// TwinCAT 3 PLC project LeakTesters
// ProgramVersion: 3.1.4024.0
// libraries:
//   Tc2_Standard, * (Beckhoff Automation GmbH)
//   Tc2_System, * (Beckhoff Automation GmbH)
//   Tc2_Utilities, * (Beckhoff Automation GmbH)
//   Tc3_EventLogger, * (Beckhoff Automation GmbH)
//   Tc3_Module, * (Beckhoff Automation GmbH)
//   VisuUserMgmt, * (System)
// project tree:
//   DUTs/ E_MachineState.TcDUT (not stored), E_StationState.TcDUT (not stored), ST_ActiveEventsHMI.TcDUT (not stored), ST_AlarmHistory.TcDUT (not stored), ST_Events.TcDUT (not stored), ST_HeightLimits.TcDUT (not stored), ST_HeightMeasurement2.TcDUT (not stored), ST_MachineStatusStruct.TcDUT (not stored), ST_MasterControlStruct.TcDUT (not stored), ST_MeasureStatistics.TcDUT (not stored), ST_Nest.TcDUT, ST_PartsInspection.TcDUT, ST_StandardStationStruct.TcDUT (not stored), ST_UserLogHMI.TcDUT (not stored)
//   DUTs/HeightMeasureFunction/ E_HeighttMeasureProcess.TcDUT (not stored)
//   DUTs/IO/ E_BoxDiag.TcDUT (not stored), E_BoxState.TcDUT (not stored), E_TerminalState.TcDUT (not stored), st_Box_Info.TcDUT (not stored), st_EL1809.TcDUT (not stored), st_EL2809.TcDUT (not stored), ST_DL_PN1.TcDUT (not stored), st_KeyenceCamera.TcDUT, st_Terminal_Info.TcDUT (not stored)
//   GVLs/ GVL_Constants.TcGVL (not stored), GVL_HMI_GLOBAL.TcGVL, GVL_IO.TcGVL, GVL_MASTER.TcGVL (not stored), GVL_PERSIST.TcGVL
//   / PlcTask.TcTTO (not stored)
//   POUs/A_Master/ Main_Master.TcPOU, PRG_FaultHandling.TcPOU, PRG_MachineStatus.TcPOU (not stored), PRG_MasterCycle.TcPOU, PRG_MasterSystemTime.TcPOU (not stored), PRG_TerminBoxInfo.TcPOU (not stored)
//   POUs/B_HightTest/ PRG_Fault_HeightTest.TcPOU (not stored), PRG_HeightTest.TcPOU
//   POUs/D_VisionTest/ PRG_Fault_VisionTest.TcPOU, PRG_VisionTest.TcPOU
//   POUs/E_HMI/ PRG_HMI.TcPOU
//   POUs/G_Utility/ FB_Alarms.TcPOU (not stored), FB_BoxInfo.TcPOU (not stored), FB_DayOfYear.TcPOU (not stored), FB_EventLog.TcPOU (not stored), FB_HeightMeasurement2.TcPOU (not stored), FB_Pulse.TcPOU (not stored), FB_TerminalInfo.TcPOU (not stored), FB_TimeControl.TcPOU (not stored), PRG_Puls.TcPOU (not stored)
//   POUs/ MAIN.TcPOU (not stored)
// real-time tasks:
//   TASK PlcTask: cycle T#10ms, priority 20, ADS port 350
// I/O:
//   DEVICE Device 1 (EtherCAT), AmsNetId 172.18.239.139.2.1
//     Term 9 (EK1100) [EK1100 EtherCAT Coupler (2A E-Bus)]
//       Term 10 (EL6070-0033) [EL6070-0033 1Ch. Licence key terminal, individual licences]
//       Term 11 (EL1809) [EL1809 16Ch. Dig. Input 24V, 3ms]
//       Term 12 (EL2809-0015) [EL2809-0015 16Ch. Dig. Output 24V DC, 0.35A, not short-circuit proof]
//       Term 13 (EL6631) [EL6631 PROFINET IO Controller]
//       Term 14 (EL9011) [EL9011 End Terminal]
//   DEVICE Device 2 (EL6631), AmsNetId 172.18.239.139.3.1
//     dl-pn1 [Keyence DL-PN1 PROFINET IO Device DL-PN1]
//       modules: Term 13 (DAP Module), Term 14 (DL-PN1), Term 15 (GT2-1.1), Term 16 (GT2-1.2), Term 17 (GT2-1.3), Term 18 (GT2-2)
//     camera-1 [KEYENCE CORPORATION. IV4-XXXX IV4-XXXX]
//       modules: Term 1 (DAP Module), Term 2 (Command Control), Term 3 (Additional Setting Value), Term 4 (Command Status Bits), Term 5 (Device Result Bits), Term 6 (Device Status Words), Term 7 (Device Statistics), Term 8 (Position Adjust Result), Term 9 (Tool Result), Term 10 (Tool Result), Term 11 (Tool Result), Term 79 (Device Result Bits)
// variable links:
//   LeakTesters/LeakTesters Instance <-> Device 1 (EtherCAT)/Term 9 (EK1100)/Term 10 (EL6070-0033)
//     PlcTask Inputs/GVL_IO.dwTerminalInfo[2].nTerminal_State <-> InfoData/State
//   LeakTesters/LeakTesters Instance <-> Device 1 (EtherCAT)/Term 9 (EK1100)/Term 11 (EL1809)
//     PlcTask Inputs/GVL_IO.dwTerminalInfo[3].nTerminal_State <-> InfoData/State
//     PlcTask Inputs/GVL_IO.dw_T02_EL1809.iCalmpClosed <-> Channel 1/Input
//     PlcTask Inputs/GVL_IO.dw_T02_EL1809.iPartPresent <-> Channel 2/Input
//   LeakTesters/LeakTesters Instance <-> Device 1 (EtherCAT)/Term 9 (EK1100)/Term 12 (EL2809-0015)
//     PlcTask Inputs/GVL_IO.dwTerminalInfo[4].nTerminal_State <-> InfoData/State
//     PlcTask Outputs/GVL_IO.dw_T03_EL2809.qEL2809_Ch3 <-> Channel 3/Output
//     PlcTask Outputs/GVL_IO.dw_T03_EL2809.qPassIndicatorGreen <-> Channel 1/Output
//     PlcTask Outputs/GVL_IO.dw_T03_EL2809.qRejectIndicatorRed <-> Channel 2/Output
//   LeakTesters/LeakTesters Instance <-> Device 1 (EtherCAT)/Term 9 (EK1100)/Term 13 (EL6631)
//     PlcTask Inputs/GVL_IO.dwTerminalInfo[5].nTerminal_State <-> InfoData/State
//   LeakTesters/LeakTesters Instance <-> Device 2 (EL6631)/camera-1
//     PlcTask Inputs/GVL_IO.dw_B06_KeyenceCamera.bBusy <-> API/Term 4 (Command Status Bits)/Subterm 6 (Command Status Bits)/Inputs/Command Status Bits Register2/Busy
//     PlcTask Inputs/GVL_IO.dw_B06_KeyenceCamera.bError <-> API/Term 4 (Command Status Bits)/Subterm 6 (Command Status Bits)/Inputs/Command Status Bits Register3/Error
//     PlcTask Inputs/GVL_IO.dw_B06_KeyenceCamera.bReady <-> API/Term 4 (Command Status Bits)/Subterm 6 (Command Status Bits)/Inputs/Command Status Bits Register2/Ready
//     PlcTask Inputs/GVL_IO.dw_B06_KeyenceCamera.bResultReady <-> API/Term 4 (Command Status Bits)/Subterm 6 (Command Status Bits)/Inputs/Command Status Bits Register2/Result_Ready
//     PlcTask Inputs/GVL_IO.dw_B06_KeyenceCamera.bRun <-> API/Term 4 (Command Status Bits)/Subterm 6 (Command Status Bits)/Inputs/Command Status Bits Register2/Run
//     PlcTask Inputs/GVL_IO.dw_B06_KeyenceCamera.bTotalResult <-> API/Term 5 (Device Result Bits)/Subterm 7 (Device Result Bits)/Inputs/Device Result Bits Register0/Total_Status
//     PlcTask Inputs/GVL_IO.dw_B06_KeyenceCamera.bTriggerFail <-> API/Term 4 (Command Status Bits)/Subterm 6 (Command Status Bits)/Inputs/Command Status Bits Register1/Trigger_Fail
//     PlcTask Outputs/GVL_IO.dw_B06_KeyenceCamera.bClearBuffer <-> API/Term 2 (Command Control)/Subterm 4 (Command Control)/Outputs/Command Control Register0/Clear_Buffer
//     PlcTask Outputs/GVL_IO.dw_B06_KeyenceCamera.bReset <-> API/Term 2 (Command Control)/Subterm 4 (Command Control)/Outputs/Command Control Register0/Clear_Warning
//     PlcTask Outputs/GVL_IO.dw_B06_KeyenceCamera.bResultReadyAck <-> API/Term 2 (Command Control)/Subterm 4 (Command Control)/Outputs/Command Control Register1/Result_Ready_Ack
//     PlcTask Outputs/GVL_IO.dw_B06_KeyenceCamera.bTrigger <-> API/Term 2 (Command Control)/Subterm 4 (Command Control)/Outputs/Command Control Register0/Trigger
//   LeakTesters/LeakTesters Instance <-> Device 2 (EL6631)/dl-pn1
//     PlcTask Inputs/GVL_IO.dwBoxInfo[17].nPnIoBoxDiag <-> Inputs/PnIoBoxDiag
//     PlcTask Inputs/GVL_IO.dwBoxInfo[17].nPnIoBoxState <-> Inputs/PnIoBoxState
//     PlcTask Inputs/GVL_IO.dw_B08_DL_PN1.dldCurrValProp <-> API/Term 14 (DL-PN1)/Subterm 23 (DL-PN1 Device)/Inputs/Sensors Status/Current_Value_Property
//     PlcTask Inputs/GVL_IO.dw_B08_DL_PN1.dldErrorStt <-> API/Term 14 (DL-PN1)/Subterm 23 (DL-PN1 Device)/Inputs/Sensors Status/Error_Status
//     PlcTask Inputs/GVL_IO.dw_B08_DL_PN1.dldExtInpResp[1] <-> API/Term 14 (DL-PN1)/Subterm 23 (DL-PN1 Device)/Inputs/External Input Response/External_Input_Response_1
//     PlcTask Inputs/GVL_IO.dw_B08_DL_PN1.dldExtInpResp[2] <-> API/Term 14 (DL-PN1)/Subterm 23 (DL-PN1 Device)/Inputs/External Input Response/External_Input_Response_2
//     PlcTask Inputs/GVL_IO.dw_B08_DL_PN1.dldExtInpResp[3] <-> API/Term 14 (DL-PN1)/Subterm 23 (DL-PN1 Device)/Inputs/External Input Response/External_Input_Response_3
//     PlcTask Inputs/GVL_IO.dw_B08_DL_PN1.dldExtInpResp[4] <-> API/Term 14 (DL-PN1)/Subterm 23 (DL-PN1 Device)/Inputs/External Input Response/External_Input_Response_4
//     PlcTask Inputs/GVL_IO.dw_B08_DL_PN1.dldExtInpResp[5] <-> API/Term 14 (DL-PN1)/Subterm 23 (DL-PN1 Device)/Inputs/External Input Response/External_Input_Response_5
//     PlcTask Inputs/GVL_IO.dw_B08_DL_PN1.dldWarningStat <-> API/Term 14 (DL-PN1)/Subterm 23 (DL-PN1 Device)/Inputs/Sensors Status/Warning_Status
//     PlcTask Inputs/GVL_IO.dw_B08_DL_PN1.gt2_1_1CurrValInv <-> API/Term 15 (GT2-1.1)/Subterm 24 (GT2-***)/Inputs/Sensor Status/Current_Value_Invalid
//     PlcTask Inputs/GVL_IO.dw_B08_DL_PN1.gt2_1_2CurrValInv <-> API/Term 16 (GT2-1.2)/Subterm 25 (GT2-***)/Inputs/Sensor Status/Current_Value_Invalid
//     PlcTask Inputs/GVL_IO.dw_B08_DL_PN1.gt2_1_3CurrValInv <-> API/Term 17 (GT2-1.3)/Subterm 26 (GT2-***)/Inputs/Sensor Status/Current_Value_Invalid
//     PlcTask Inputs/GVL_IO.dw_B08_DL_PN1.gt2_1_1CurrValOvrR <-> API/Term 15 (GT2-1.1)/Subterm 24 (GT2-***)/Inputs/Sensor Status/Current_Value_Over_Range
//     PlcTask Inputs/GVL_IO.dw_B08_DL_PN1.gt2_1_2CurrValOvrR <-> API/Term 16 (GT2-1.2)/Subterm 25 (GT2-***)/Inputs/Sensor Status/Current_Value_Over_Range
//     PlcTask Inputs/GVL_IO.dw_B08_DL_PN1.gt2_1_3CurrValOvrR <-> API/Term 17 (GT2-1.3)/Subterm 26 (GT2-***)/Inputs/Sensor Status/Current_Value_Over_Range
//     PlcTask Inputs/GVL_IO.dw_B08_DL_PN1.gt2_1_1CurrValUndR <-> API/Term 15 (GT2-1.1)/Subterm 24 (GT2-***)/Inputs/Sensor Status/Current_Value_Under_Range
//     PlcTask Inputs/GVL_IO.dw_B08_DL_PN1.gt2_1_2CurrValUndR <-> API/Term 16 (GT2-1.2)/Subterm 25 (GT2-***)/Inputs/Sensor Status/Current_Value_Under_Range
//     PlcTask Inputs/GVL_IO.dw_B08_DL_PN1.gt2_1_3CurrValUndR <-> API/Term 17 (GT2-1.3)/Subterm 26 (GT2-***)/Inputs/Sensor Status/Current_Value_Under_Range
//     PlcTask Inputs/GVL_IO.dw_B08_DL_PN1.gt2_1_1CurrentValue <-> API/Term 15 (GT2-1.1)/Subterm 24 (GT2-***)/Inputs/Current Value
//     PlcTask Inputs/GVL_IO.dw_B08_DL_PN1.gt2_1_2CurrentValue <-> API/Term 16 (GT2-1.2)/Subterm 25 (GT2-***)/Inputs/Current Value
//     PlcTask Inputs/GVL_IO.dw_B08_DL_PN1.gt2_1_3CurrentValue <-> API/Term 17 (GT2-1.3)/Subterm 26 (GT2-***)/Inputs/Current Value
//     PlcTask Inputs/GVL_IO.dw_B08_DL_PN1.gt2_1_1ErrorStat <-> API/Term 15 (GT2-1.1)/Subterm 24 (GT2-***)/Inputs/Sensor Status/Error_Status
//     PlcTask Inputs/GVL_IO.dw_B08_DL_PN1.gt2_1_2ErrorStat <-> API/Term 16 (GT2-1.2)/Subterm 25 (GT2-***)/Inputs/Sensor Status/Error_Status
//     PlcTask Inputs/GVL_IO.dw_B08_DL_PN1.gt2_1_3ErrorStat <-> API/Term 17 (GT2-1.3)/Subterm 26 (GT2-***)/Inputs/Sensor Status/Error_Status
//     PlcTask Inputs/GVL_IO.dw_B08_DL_PN1.gt2_1_1ExtInpRes[1] <-> API/Term 15 (GT2-1.1)/Subterm 24 (GT2-***)/Inputs/External Input Response/External_Input_Response_1
//     PlcTask Inputs/GVL_IO.dw_B08_DL_PN1.gt2_1_1ExtInpRes[2] <-> API/Term 15 (GT2-1.1)/Subterm 24 (GT2-***)/Inputs/External Input Response/External_Input_Response_2
//     PlcTask Inputs/GVL_IO.dw_B08_DL_PN1.gt2_1_1ExtInpRes[3] <-> API/Term 15 (GT2-1.1)/Subterm 24 (GT2-***)/Inputs/External Input Response/External_Input_Response_3
//     PlcTask Inputs/GVL_IO.dw_B08_DL_PN1.gt2_1_1ExtInpRes[4] <-> API/Term 15 (GT2-1.1)/Subterm 24 (GT2-***)/Inputs/External Input Response/External_Input_Response_4
//     PlcTask Inputs/GVL_IO.dw_B08_DL_PN1.gt2_1_1ExtInpRes[5] <-> API/Term 15 (GT2-1.1)/Subterm 24 (GT2-***)/Inputs/External Input Response/External_Input_Response_5
//     PlcTask Inputs/GVL_IO.dw_B08_DL_PN1.gt2_1_2ExtInpRes[1] <-> API/Term 16 (GT2-1.2)/Subterm 25 (GT2-***)/Inputs/External Input Response/External_Input_Response_1
//     PlcTask Inputs/GVL_IO.dw_B08_DL_PN1.gt2_1_2ExtInpRes[2] <-> API/Term 16 (GT2-1.2)/Subterm 25 (GT2-***)/Inputs/External Input Response/External_Input_Response_2
//     PlcTask Inputs/GVL_IO.dw_B08_DL_PN1.gt2_1_2ExtInpRes[3] <-> API/Term 16 (GT2-1.2)/Subterm 25 (GT2-***)/Inputs/External Input Response/External_Input_Response_3
//     PlcTask Inputs/GVL_IO.dw_B08_DL_PN1.gt2_1_2ExtInpRes[4] <-> API/Term 16 (GT2-1.2)/Subterm 25 (GT2-***)/Inputs/External Input Response/External_Input_Response_4
//     PlcTask Inputs/GVL_IO.dw_B08_DL_PN1.gt2_1_2ExtInpRes[5] <-> API/Term 16 (GT2-1.2)/Subterm 25 (GT2-***)/Inputs/External Input Response/External_Input_Response_5
//     PlcTask Inputs/GVL_IO.dw_B08_DL_PN1.gt2_1_3ExtInpRes[1] <-> API/Term 17 (GT2-1.3)/Subterm 26 (GT2-***)/Inputs/External Input Response/External_Input_Response_1
//     PlcTask Inputs/GVL_IO.dw_B08_DL_PN1.gt2_1_3ExtInpRes[2] <-> API/Term 17 (GT2-1.3)/Subterm 26 (GT2-***)/Inputs/External Input Response/External_Input_Response_2
//     PlcTask Inputs/GVL_IO.dw_B08_DL_PN1.gt2_1_3ExtInpRes[3] <-> API/Term 17 (GT2-1.3)/Subterm 26 (GT2-***)/Inputs/External Input Response/External_Input_Response_3
//     PlcTask Inputs/GVL_IO.dw_B08_DL_PN1.gt2_1_3ExtInpRes[4] <-> API/Term 17 (GT2-1.3)/Subterm 26 (GT2-***)/Inputs/External Input Response/External_Input_Response_4
//     PlcTask Inputs/GVL_IO.dw_B08_DL_PN1.gt2_1_3ExtInpRes[5] <-> API/Term 17 (GT2-1.3)/Subterm 26 (GT2-***)/Inputs/External Input Response/External_Input_Response_5
//     PlcTask Inputs/GVL_IO.dw_B08_DL_PN1.gt2_1_1Output[1] <-> API/Term 15 (GT2-1.1)/Subterm 24 (GT2-***)/Inputs/Sensor Outputs/Output_1
//     PlcTask Inputs/GVL_IO.dw_B08_DL_PN1.gt2_1_1Output[2] <-> API/Term 15 (GT2-1.1)/Subterm 24 (GT2-***)/Inputs/Sensor Outputs/Output_2
//     PlcTask Inputs/GVL_IO.dw_B08_DL_PN1.gt2_1_1Output[3] <-> API/Term 15 (GT2-1.1)/Subterm 24 (GT2-***)/Inputs/Sensor Outputs/Output_3
//     PlcTask Inputs/GVL_IO.dw_B08_DL_PN1.gt2_1_1Output[4] <-> API/Term 15 (GT2-1.1)/Subterm 24 (GT2-***)/Inputs/Sensor Outputs/Output_4
//     PlcTask Inputs/GVL_IO.dw_B08_DL_PN1.gt2_1_1Output[5] <-> API/Term 15 (GT2-1.1)/Subterm 24 (GT2-***)/Inputs/Sensor Outputs/Output_5
//     PlcTask Inputs/GVL_IO.dw_B08_DL_PN1.gt2_1_2Output[1] <-> API/Term 16 (GT2-1.2)/Subterm 25 (GT2-***)/Inputs/Sensor Outputs/Output_1
//     PlcTask Inputs/GVL_IO.dw_B08_DL_PN1.gt2_1_2Output[2] <-> API/Term 16 (GT2-1.2)/Subterm 25 (GT2-***)/Inputs/Sensor Outputs/Output_2
//     PlcTask Inputs/GVL_IO.dw_B08_DL_PN1.gt2_1_2Output[3] <-> API/Term 16 (GT2-1.2)/Subterm 25 (GT2-***)/Inputs/Sensor Outputs/Output_3
//     PlcTask Inputs/GVL_IO.dw_B08_DL_PN1.gt2_1_2Output[4] <-> API/Term 16 (GT2-1.2)/Subterm 25 (GT2-***)/Inputs/Sensor Outputs/Output_4
//     PlcTask Inputs/GVL_IO.dw_B08_DL_PN1.gt2_1_2Output[5] <-> API/Term 16 (GT2-1.2)/Subterm 25 (GT2-***)/Inputs/Sensor Outputs/Output_5
//     PlcTask Inputs/GVL_IO.dw_B08_DL_PN1.gt2_1_3Output[1] <-> API/Term 17 (GT2-1.3)/Subterm 26 (GT2-***)/Inputs/Sensor Outputs/Output_1
//     PlcTask Inputs/GVL_IO.dw_B08_DL_PN1.gt2_1_3Output[2] <-> API/Term 17 (GT2-1.3)/Subterm 26 (GT2-***)/Inputs/Sensor Outputs/Output_2
//     PlcTask Inputs/GVL_IO.dw_B08_DL_PN1.gt2_1_3Output[3] <-> API/Term 17 (GT2-1.3)/Subterm 26 (GT2-***)/Inputs/Sensor Outputs/Output_3
//     PlcTask Inputs/GVL_IO.dw_B08_DL_PN1.gt2_1_3Output[4] <-> API/Term 17 (GT2-1.3)/Subterm 26 (GT2-***)/Inputs/Sensor Outputs/Output_4
//     PlcTask Inputs/GVL_IO.dw_B08_DL_PN1.gt2_1_3Output[5] <-> API/Term 17 (GT2-1.3)/Subterm 26 (GT2-***)/Inputs/Sensor Outputs/Output_5
//     PlcTask Inputs/GVL_IO.dw_B08_DL_PN1.gt2_1_1WarningStat <-> API/Term 15 (GT2-1.1)/Subterm 24 (GT2-***)/Inputs/Sensor Status/Warning_Status
//     PlcTask Inputs/GVL_IO.dw_B08_DL_PN1.gt2_1_2WarningStat <-> API/Term 16 (GT2-1.2)/Subterm 25 (GT2-***)/Inputs/Sensor Status/Warning_Status
//     PlcTask Inputs/GVL_IO.dw_B08_DL_PN1.gt2_1_3WarningStat <-> API/Term 17 (GT2-1.3)/Subterm 26 (GT2-***)/Inputs/Sensor Status/Warning_Status
//     PlcTask Inputs/GVL_IO.dw_B08_DL_PN1.gt2_2CurrValInv <-> API/Term 18 (GT2-2)/Subterm 27 (GT2-***)/Inputs/Sensor Status/Current_Value_Invalid
//     PlcTask Inputs/GVL_IO.dw_B08_DL_PN1.gt2_2CurrValOvrR <-> API/Term 18 (GT2-2)/Subterm 27 (GT2-***)/Inputs/Sensor Status/Current_Value_Over_Range
//     PlcTask Inputs/GVL_IO.dw_B08_DL_PN1.gt2_2CurrValUndR <-> API/Term 18 (GT2-2)/Subterm 27 (GT2-***)/Inputs/Sensor Status/Current_Value_Under_Range
//     PlcTask Inputs/GVL_IO.dw_B08_DL_PN1.gt2_2CurrentValue <-> API/Term 18 (GT2-2)/Subterm 27 (GT2-***)/Inputs/Current Value
//     PlcTask Inputs/GVL_IO.dw_B08_DL_PN1.gt2_2ErrorStat <-> API/Term 18 (GT2-2)/Subterm 27 (GT2-***)/Inputs/Sensor Status/Error_Status
//     PlcTask Inputs/GVL_IO.dw_B08_DL_PN1.gt2_2ExtInpRes[1] <-> API/Term 18 (GT2-2)/Subterm 27 (GT2-***)/Inputs/External Input Response/External_Input_Response_1
//     PlcTask Inputs/GVL_IO.dw_B08_DL_PN1.gt2_2ExtInpRes[2] <-> API/Term 18 (GT2-2)/Subterm 27 (GT2-***)/Inputs/External Input Response/External_Input_Response_2
//     PlcTask Inputs/GVL_IO.dw_B08_DL_PN1.gt2_2ExtInpRes[3] <-> API/Term 18 (GT2-2)/Subterm 27 (GT2-***)/Inputs/External Input Response/External_Input_Response_3
//     PlcTask Inputs/GVL_IO.dw_B08_DL_PN1.gt2_2ExtInpRes[4] <-> API/Term 18 (GT2-2)/Subterm 27 (GT2-***)/Inputs/External Input Response/External_Input_Response_4
//     PlcTask Inputs/GVL_IO.dw_B08_DL_PN1.gt2_2ExtInpRes[5] <-> API/Term 18 (GT2-2)/Subterm 27 (GT2-***)/Inputs/External Input Response/External_Input_Response_5
//     PlcTask Inputs/GVL_IO.dw_B08_DL_PN1.gt2_2Output[1] <-> API/Term 18 (GT2-2)/Subterm 27 (GT2-***)/Inputs/Sensor Outputs/Output_1
//     PlcTask Inputs/GVL_IO.dw_B08_DL_PN1.gt2_2Output[2] <-> API/Term 18 (GT2-2)/Subterm 27 (GT2-***)/Inputs/Sensor Outputs/Output_2
//     PlcTask Inputs/GVL_IO.dw_B08_DL_PN1.gt2_2Output[3] <-> API/Term 18 (GT2-2)/Subterm 27 (GT2-***)/Inputs/Sensor Outputs/Output_3
//     PlcTask Inputs/GVL_IO.dw_B08_DL_PN1.gt2_2Output[4] <-> API/Term 18 (GT2-2)/Subterm 27 (GT2-***)/Inputs/Sensor Outputs/Output_4
//     PlcTask Inputs/GVL_IO.dw_B08_DL_PN1.gt2_2Output[5] <-> API/Term 18 (GT2-2)/Subterm 27 (GT2-***)/Inputs/Sensor Outputs/Output_5
//     PlcTask Inputs/GVL_IO.dw_B08_DL_PN1.gt2_2WarningStat <-> API/Term 18 (GT2-2)/Subterm 27 (GT2-***)/Inputs/Sensor Status/Warning_Status
//     PlcTask Outputs/GVL_IO.dw_B08_DL_PN1.dldExtInpRespOut[1] <-> API/Term 14 (DL-PN1)/Subterm 23 (DL-PN1 Device)/Outputs/External Input Requests/External_Input_Request_1
//     PlcTask Outputs/GVL_IO.dw_B08_DL_PN1.dldExtInpRespOut[2] <-> API/Term 14 (DL-PN1)/Subterm 23 (DL-PN1 Device)/Outputs/External Input Requests/External_Input_Request_2
//     PlcTask Outputs/GVL_IO.dw_B08_DL_PN1.dldExtInpRespOut[3] <-> API/Term 14 (DL-PN1)/Subterm 23 (DL-PN1 Device)/Outputs/External Input Requests/External_Input_Request_3
//     PlcTask Outputs/GVL_IO.dw_B08_DL_PN1.dldExtInpRespOut[4] <-> API/Term 14 (DL-PN1)/Subterm 23 (DL-PN1 Device)/Outputs/External Input Requests/External_Input_Request_4
//     PlcTask Outputs/GVL_IO.dw_B08_DL_PN1.dldExtInpRespOut[5] <-> API/Term 14 (DL-PN1)/Subterm 23 (DL-PN1 Device)/Outputs/External Input Requests/External_Input_Request_5
//     PlcTask Outputs/GVL_IO.dw_B08_DL_PN1.gt2_1_1ExtInpResOut[1] <-> API/Term 15 (GT2-1.1)/Subterm 24 (GT2-***)/Outputs/External Input Requests/External_Input_Request_1
//     PlcTask Outputs/GVL_IO.dw_B08_DL_PN1.gt2_1_1ExtInpResOut[2] <-> API/Term 15 (GT2-1.1)/Subterm 24 (GT2-***)/Outputs/External Input Requests/External_Input_Request_2
//     PlcTask Outputs/GVL_IO.dw_B08_DL_PN1.gt2_1_1ExtInpResOut[3] <-> API/Term 15 (GT2-1.1)/Subterm 24 (GT2-***)/Outputs/External Input Requests/External_Input_Request_3
//     PlcTask Outputs/GVL_IO.dw_B08_DL_PN1.gt2_1_1ExtInpResOut[4] <-> API/Term 15 (GT2-1.1)/Subterm 24 (GT2-***)/Outputs/External Input Requests/External_Input_Request_4
//     PlcTask Outputs/GVL_IO.dw_B08_DL_PN1.gt2_1_1ExtInpResOut[5] <-> API/Term 15 (GT2-1.1)/Subterm 24 (GT2-***)/Outputs/External Input Requests/External_Input_Request_5
//     PlcTask Outputs/GVL_IO.dw_B08_DL_PN1.gt2_1_2ExtInpResOut[1] <-> API/Term 16 (GT2-1.2)/Subterm 25 (GT2-***)/Outputs/External Input Requests/External_Input_Request_1
//     PlcTask Outputs/GVL_IO.dw_B08_DL_PN1.gt2_1_2ExtInpResOut[2] <-> API/Term 16 (GT2-1.2)/Subterm 25 (GT2-***)/Outputs/External Input Requests/External_Input_Request_2
//     PlcTask Outputs/GVL_IO.dw_B08_DL_PN1.gt2_1_2ExtInpResOut[3] <-> API/Term 16 (GT2-1.2)/Subterm 25 (GT2-***)/Outputs/External Input Requests/External_Input_Request_3
//     PlcTask Outputs/GVL_IO.dw_B08_DL_PN1.gt2_1_2ExtInpResOut[4] <-> API/Term 16 (GT2-1.2)/Subterm 25 (GT2-***)/Outputs/External Input Requests/External_Input_Request_4
//     PlcTask Outputs/GVL_IO.dw_B08_DL_PN1.gt2_1_2ExtInpResOut[5] <-> API/Term 16 (GT2-1.2)/Subterm 25 (GT2-***)/Outputs/External Input Requests/External_Input_Request_5
//     PlcTask Outputs/GVL_IO.dw_B08_DL_PN1.gt2_1_3ExtInpResOut[1] <-> API/Term 17 (GT2-1.3)/Subterm 26 (GT2-***)/Outputs/External Input Requests/External_Input_Request_1
//     PlcTask Outputs/GVL_IO.dw_B08_DL_PN1.gt2_1_3ExtInpResOut[2] <-> API/Term 17 (GT2-1.3)/Subterm 26 (GT2-***)/Outputs/External Input Requests/External_Input_Request_2
//     PlcTask Outputs/GVL_IO.dw_B08_DL_PN1.gt2_1_3ExtInpResOut[3] <-> API/Term 17 (GT2-1.3)/Subterm 26 (GT2-***)/Outputs/External Input Requests/External_Input_Request_3
//     PlcTask Outputs/GVL_IO.dw_B08_DL_PN1.gt2_1_3ExtInpResOut[4] <-> API/Term 17 (GT2-1.3)/Subterm 26 (GT2-***)/Outputs/External Input Requests/External_Input_Request_4
//     PlcTask Outputs/GVL_IO.dw_B08_DL_PN1.gt2_1_3ExtInpResOut[5] <-> API/Term 17 (GT2-1.3)/Subterm 26 (GT2-***)/Outputs/External Input Requests/External_Input_Request_5
//     PlcTask Outputs/GVL_IO.dw_B08_DL_PN1.gt2_2ExtInpResOut[1] <-> API/Term 18 (GT2-2)/Subterm 27 (GT2-***)/Outputs/External Input Requests/External_Input_Request_1
//     PlcTask Outputs/GVL_IO.dw_B08_DL_PN1.gt2_2ExtInpResOut[2] <-> API/Term 18 (GT2-2)/Subterm 27 (GT2-***)/Outputs/External Input Requests/External_Input_Request_2
//     PlcTask Outputs/GVL_IO.dw_B08_DL_PN1.gt2_2ExtInpResOut[3] <-> API/Term 18 (GT2-2)/Subterm 27 (GT2-***)/Outputs/External Input Requests/External_Input_Request_3
//     PlcTask Outputs/GVL_IO.dw_B08_DL_PN1.gt2_2ExtInpResOut[4] <-> API/Term 18 (GT2-2)/Subterm 27 (GT2-***)/Outputs/External Input Requests/External_Input_Request_4
//     PlcTask Outputs/GVL_IO.dw_B08_DL_PN1.gt2_2ExtInpResOut[5] <-> API/Term 18 (GT2-2)/Subterm 27 (GT2-***)/Outputs/External Input Requests/External_Input_Request_5

// ---- DUTs/IO/st_KeyenceCamera.TcDUT
TYPE st_KeyenceCamera :
STRUCT
	
	////////////////////////////////////////////////////INPUTS//////////////////////////////////////////////////

	bResultReady							AT%I*					: BOOL;
	bError									AT%I*					: BOOL;
	bBusy									AT%I*					: BOOL;
	bRun									AT%I*					: BOOL;
	bReady									AT%I*					: BOOL;
	bTotalResult							AT%I*					: BOOL;
	bTriggerFail							AT%I*					: BOOL;
	
	////////////////////////////////////////////////////OUTPUTS//////////////////////////////////////////////////
	
	bTrigger								AT%Q*					: BOOL;//
	bReset									AT%Q*					: BOOL;//
	bResultReadyAck							AT%Q*					: BOOL;//
	bClearBuffer							AT%Q*					: BOOL;//

END_STRUCT
END_TYPE

// ---- DUTs/ST_Nest.TcDUT
TYPE ST_Nest :
STRUCT
		 

	 
     bNestPartProced    : BOOL;
     bNestPartOK        : BOOL;
	 bNestPresent       : BOOL;

	 
	 bHeightPass		: BOOL;
	 bVisionPass		: BOOL;
	 bPiecePass			: BOOL;
	 
	 bHeightReject		: BOOL;
	 bVisionReject		: BOOL;	
	 bPieceReject		: BOOL; 
	 
	 sHeightHMI			: WSTRING;
	 sVisionHMI			: WSTRING;
	 sPieceHMI			: WSTRING;

	 nDistance			: ARRAY[1..3] OF REAL;
	 nTarget			: ARRAY[1..3] OF REAL;	

 
	 sDate				: STRING;
	 sTime				: STRING;

END_STRUCT
END_TYPE

// ---- DUTs/ST_PartsInspection.TcDUT
TYPE ST_PartsInspection :
STRUCT
	
	nVisionPartsGood				: DINT;
	nVisionTotalPartsGood			: DINT;
	nVisionPartsFailed				: DINT;
	nVisionTotalPartsFailed			: DINT;
	
	nHeightPartsGood				: DINT;
	nHeightTotalPartsGood			: DINT;
	nHeightPartsFailed				: DINT;
	nHeightTotalPartsFailed			: DINT;
	
	nHeightDistancePartsGood		: ARRAY[1..4] OF DINT;
	nHeightDistanceTotalPartsGood	: ARRAY[1..4] OF DINT;
	nHeightDistancePartsFailed		: ARRAY[1..4] OF DINT;
	nHeightDistanceTotalPartsFailed	: ARRAY[1..4] OF DINT;
	
	nPartsGood						: DINT;
	nTotalPartsGood					: DINT;
	nPartsFailed					: DINT;
	nTotalPartsFailed				: DINT;					
	
	bPartok							: BOOL;
	bPartFail						: BOOL;
END_STRUCT
END_TYPE

// ---- GVLs/GVL_HMI_GLOBAL.TcGVL
{attribute 'qualified_only'}
VAR_GLOBAL
	
	//User Log, Shut down, Quit HMI
	bQuitHmi						: BOOL;
	sUserGroup						: STRING;
	sUserGroup2						: STRING;
	sUserName						: STRING;
	bLogOut							: BOOL;
	bUserLogedIntSignal				: BOOL;
	bShutDown						: BOOL;

	//General
	bStopButton						: BOOL;
	bStartButton					: BOOL;
	bResetButton					: BOOL;
	nRegionMain						: INT;
	bResetGoodParts					: BOOL;
	bResetFailedParts				: BOOL;
	
	aEventTexts						: ARRAY [0..767] OF T_MaxSTring; //Event texts - set only once
	bEventTextsSet					: BOOL;
	aEventFlags						: ARRAY [0..767] OF BOOL;		//All event states combined from master na stations
	aActiveEvents					: ARRAY [0..39] OF T_MaxSTring;	//Active events - connected to Alarm scree in HMI	
	stActiveEventsHMI				: ARRAY [0..39] OF ST_ActiveEventsHMI;
	
	sMessageToOperator				: WSTRING(200);
	sActualProcess					: WSTRING(200);
	aIOScreen						: ARRAY [0..8] OF STRING(200);
	aManualScreen					: ARRAY [0..1] OF STRING(200);
	bResetPassAndFail				: BOOL;
	bEnableManualMode				: BOOL;
	bRejectPieceAcknowledge			: BOOL;
	bRejectPieceDialogTrig			: BOOL;
	bAutocycleFaultDialog			: BOOL;
	
	
	
	// ------ Screen Info / Data -----------	
	sSystemDate					: STRING;
	sSystemTime					: STRING;
	ntAMSNetID					: T_AmsNetId := '172.18.239.139.1.1';
	
	
	
	//Camera
	bManualModeOff					: ARRAY[1..2] OF BOOL;
	bVisionPass						: BOOL;
	bResetVisionGoodParts			: BOOL;
	bResetVisionBadParts			: BOOL;
	
	//Height Tester
	bHeightTestPass					: BOOL;
	bResetHeightGoodParts			: BOOL;
	bResetHeightFailParts			: BOOL;
	bManualHeightTrigger			: BOOL;
	aResetHeightSensorGoodParts		: ARRAY[1..4] OF BOOL;
	aResetHeightSensorBadParts		: ARRAY[1..4] OF BOOL;
	
	
	bSetSetPointsHeightTest			: BOOL;
	bManualMeasureHeightTest		: BOOL;
	aGeneralPassHeightTest			: ARRAY[1..5] OF BOOL;
	aGeneralFailHeightTest			: ARRAY[1..5] OF BOOL;
	
	anValueScaledHeightTest			: ARRAY[1..4] OF DINT;
	
	aSensorSetPointsHeightTest		: ARRAY[1..4] OF DINT;
	
	nHeightMeasureStateValue		: ARRAY[1..4] OF DINT;
	bProbesPositionOk				: BOOL;
	

	

	
	

END_VAR
VAR_GLOBAL PERSISTENT
	
	aStatistics					: ARRAY [1..201] OF ST_Nest;//LA** 04092025 >> : ARRAY [1..200] OF ST_Nest;
	stAlarmHistory				:ARRAY [00..250] OF ST_AlarmHistory;
	aEventLog					:ARRAY [0..250] OF T_MaxSTring;	//Event log - connected to alarm history in HMI	
	aTimeLog					:ARRAY [0..250] OF T_MaxSTring;
	aDateLog					:ARRAY [0..250] OF T_MaxSTring;
	aMinLimitHeightTest				: ARRAY[1..4] OF DINT;
	aMaxLimitHeightTest				: ARRAY[1..4] OF DINT;	
		
END_VAR

// ---- GVLs/GVL_IO.TcGVL
{attribute 'qualified_only'}
VAR_GLOBAL
	
    //--------------------------------------------------------------------------------------------------------

    dwTerminalInfo                                          : ARRAY[0..20] OF  st_Terminal_Info; // all terminal's status information 
	dwBoxInfo                                               : ARRAY[15..17] OF st_Box_Info;//Camera, Leak, Height
	//--------------------------------------------------------------------------------------------------------
	
	(* Terminal *)
	
	//	dw_T01_EK1100                                                	| EtherCAT Coupler 
	//	dw_T02_EL6070-0033                                           	| EtherCAT Terminal, license key for TwinCAT 3.1
	
	dw_T02_EL1809                                                		: st_EL1809; //16 Channel Digital Input ( 24VDC ) 
	dw_T03_EL2809                                                		: st_EL2809; // 16 Channel Digital Output ( 24VDC )
	//dw_T04_EL6631                                                	| EtherCAT Terminal, 2-port communication interface, PROFINET RT, controller - Data for Box's MDU1020 and SR2000W
 	//  dw_T05_EL9011                                                	| Bus end cover for E-bus contacts
	dw_B06_KeyenceCamera                                             	: st_KeyenceCamera;
		
	dw_B08_DL_PN1                                                		: ST_DL_PN1; // Keyence GT2 Position Sensors 
	
	
END_VAR

// ---- GVLs/GVL_PERSIST.TcGVL
{attribute 'qualified_only'}
VAR_GLOBAL PERSISTENT
	
stPartsInspection			: ST_PartsInspection;
stUserLogHMI				: ARRAY[0..250] OF ST_UserLogHMI;
UserId						: UINT;
nCycleNumber				: INT;

aSensorSetPointsHeightTest		: ARRAY[1..4] OF DINT;
aTolerancesHeightTest			: ARRAY[1..4] OF DINT;

stHeightLimits					: ST_HeightLimits;





	
	
END_VAR

// ---- POUs/A_Master/Main_Master.TcPOU
PROGRAM Main_Master
VAR
	i                       :INT; //Int to handle user log index	
	k						:INT; //Int to handle user log index
	j						:INT;
	l						:INT;
	
	//////UserLog
	
	sUserGroupID			:	STRING;
	nSize					:	UDINT					:=9;
	nLen					:	UDINT					:=18;
	npos					:	UDINT					:=1;
	tonUserLogOut           :	Tc2_Standard.TON;
	fbStringFormatter       :	Tc2_Utilities.FB_FormatString;
	fbEventLogger			:	FB_EventLog;
	rUserLoggedIn			: 	R_TRIG;
	tUserLoggedIn			: 	TON;
	bFirstScan				:   BOOL;
	tFirstScan				:   TON;

	bUserLoggedIn			: 	BOOL;
	

	
	
	/////ShutDown&Quit
	closeChrome 			: 	NT_StartProcess;	
	ntShutdown					: TC2_Utilities.NT_Shutdown;
	ntError						: BOOL;
	ntBusy						: BOOL;
	ntErrorID					: UDINT;

	
	
	/////General

END_VAR

 PRG_FaultHandling(aAlarms := GVL_Master.stAlarms );
PRG_Fault_HeightTest(aAlarms := GVL_Master.stAlarms);
PRG_Fault_VisionTest(aAlarms := GVL_Master.stAlarms);

PRG_MachineStatus();
PRG_MasterCycle(stStationStruct:= GVL_Master.stStationSruct[0]);
PRG_MasterSystemTime();
ACT_ShutdownAndQuit();
ACT_UserLog();
MapUnitEventsToHmi();
PRG_HMI();
PRG_Puls();
ACT_FirstScan();
PRG_TerminBoxInfo();

//Stations
PRG_HeightTest(stStationStruct:= GVL_Master.stStationSruct[1]);
PRG_VisionTest(stStationStruct:= GVL_Master.stStationSruct[3]);



fbEventLogger(	bEnable       	:= PRG_MasterSystemTime.bReadyToRead AND GVL_MASTER.stMasterControl.bPowerUpTimerComplete,
			    sDateTime     	:= PRG_MasterSystemTime.sDateTimeSpaces,
			    aEventFlags   	:= GVL_HMI_GLOBAL.aEventFlags,
			    aEventTexts   	:= GVL_HMI_GLOBAL.aEventTexts,
			    aActiveEvents 	:= GVL_HMI_GLOBAL.aActiveEvents,
			    aEventLog     	:= GVL_HMI_GLOBAL.aEventLog,
				siDate			:= GVL_HMI_GLOBAL.sSystemDate,
				siTime			:= GVL_HMI_GLOBAL.sSystemTime,
				soDate			:= GVL_HMI_GLOBAL.aDateLog,
				soTime			:= GVL_HMI_GLOBAL.aTimeLog
);



 

IF GVL_MASTER.bFlashScale THEN
FOR j := 0 TO 39 DO
	
GVL_HMI_GLOBAL.stActiveEventsHMI[j].sActiveEvents := GVL_HMI_GLOBAL.aActiveEvents[j];
END_FOR
FOR l:=0 TO 250 DO
	
	GVL_HMI_GLOBAL.stAlarmHistory[l].sEventlog 	:= GVL_HMI_GLOBAL.aEventLog[l];
	GVL_HMI_GLOBAL.stAlarmHistory[l].sDate		:= GVL_HMI_GLOBAL.aDateLog[l];
	GVL_HMI_GLOBAL.stAlarmHistory[l].sTime		:= GVL_HMI_GLOBAL.aTimeLog[l];
END_FOR
ELSE 
	
j:=0; 
l:=0;

END_IF

ACTION ACT_FirstScan:
tFirstScan(IN := NOT bFirstScan, PT := T#5S);
END_ACTION

ACTION ACT_ShutdownAndQuit:
closeChrome(
    NetId := '',
    PathStr := 'C:\Windows\System32\mshta vbscript:Execute("CreateObject(""WScript.Shell"").Run ""powershell -c',
    DirName := 'C:\Windows\System32\WindowsPowerShell\v1.0',
    ComndLine := 'taskkill /F /IM chrome.exe /T"", 0: window.close")',
    Start := GVL_HMI_GLOBAL.bQuitHmi,
    TmOut := DEFAULT_ADS_TIMEOUT
);
 
GVL_HMI_GLOBAL.bQuitHmi:= FALSE;

ntShutdown(NETID := GVL_HMI_GLOBAL.ntAMSNetID, DELAY := 5, START := GVL_HMI_GLOBAL.bShutDown, BUSY => ntBusy, ERR => ntError, ERRID => ntErrorID);
END_ACTION

ACTION ACT_UserLog:

//Getting user group

Tc2_Utilities.DELETE2( ADR(GVL_HMI_GLOBAL.sUserGroup), ADR(sUserGroupID), NSize, Nlen, nPos) ;

IF sUserGroupID = 'Administ' THEN
	
	GVL_HMI_GLOBAL.sUserGroup2 := 'Administrator';

ELSE GVL_HMI_GLOBAL.sUserGroup2 := sUserGroupID;
	

END_IF


//Logout 

tonUserLogOut( IN := (sUserGroupID = 'Administ' OR sUserGroupID ='Engineer') AND GVL_HMI_GLOBAL.bUserLogedIntSignal , PT := T#10M);

IF tonUserLogOut.Q AND (sUserGroupID = 'Administ' OR sUserGroupID ='Engineer') THEN
	
	GVL_HMI_GLOBAL.bLogOut 	:= TRUE;

	ELSE GVL_HMI_GLOBAL.bLogOut := FALSE;

END_IF

tUserLoggedIn( IN := GVL_HMI_GLOBAL.bUserLogedIntSignal, PT := T#2S);

rUserLoggedIn( CLK := tUserLoggedIn.Q);


IF rUserLoggedIn.Q THEN
	
	FOR i :=200 TO 1 BY (-1) DO
		GVL_PERSIST.stUserLogHMI[i]	:= GVL_PERSIST.stUserLogHMI[i-1];
	END_FOR
	
	GVL_PERSIST.stUserLogHMI[0].UserLog := GVL_HMI_GLOBAL.sUserName;
	GVL_PERSIST.stUserLogHMI[0].UserLogTime := GVL_HMI_GLOBAL.sSystemTime;
	GVL_PERSIST.stUserLogHMI[0].UserLogDate := GVL_HMI_GLOBAL.sSystemDate;

END_IF
END_ACTION

METHOD MapUnitEventsToHMI : BOOL
VAR_INPUT
END_VAR

VAR
	i		:INT; 	//Unit index
	j		:INT;	//Unit event index
	k		:INT; 	//HMI event index	
END_VAR
//Set event texts first
IF GVL_Master.stAlarms[0].bEventTextsSet AND
   GVL_Master.stAlarms[1].bEventTextsSet AND
   GVL_Master.stAlarms[3].bEventTextsSet AND
   NOT GVL_HMI_GLOBAL.bEventTextsSet 
THEN
	SetEventTexts();
		
	GVL_HMI_GLOBAL.bEventTextsSet := TRUE;
END_IF

//Map events from master and stations into HMI events
IF GVL_HMI_GLOBAL.bEventTextsSet THEN
	k := 0; 
	FOR i := 0 TO 3 DO
		FOR j := 0 TO 128 - 1 DO
			GVL_HMI_GLOBAL.aEventFlags[k] := GVL_Master.stAlarms[i].aEventFlags[j];
			k := k + 1;
		END_FOR
	END_FOR
END_IF
END_METHOD

METHOD SetEventTexts : BOOL
VAR_INPUT
END_VAR
VAR
	i				:INT; 	//Unit index
	j				:INT;	//HMI event index
	k				:INT;	//
END_VAR
//Set global event texts based on unit event texts (master and stations
k := 0;
FOR i := 0 TO 3 DO
	//For each unit (master, station1, station2)
	//Alarm texts
	FOR j := 0 TO 99 DO
		fbStringFormatter(	sFormat := 'Alarm No. %d - %s', 
					 	arg1 := F_INT(k), 
						arg2 := F_String(GVL_Master.stAlarms[i].aEventTexts[j]),
						sOut => GVL_HMI_GLOBAL.aEventTexts[k]);
						
		k := k + 1; //Increment global events index
	END_FOR
	
	//Messages
	FOR j := 100 TO 127 DO
		fbStringFormatter(	sFormat := 'Message No. %d - %s', 
					 		arg1 := F_INT(k), 
							arg2 := F_String(GVL_Master.stAlarms[i].aEventTexts[j]),
							sOut => GVL_HMI_GLOBAL.aEventTexts[k]);
							
		k := k + 1; //Increment global events index
	END_FOR
END_FOR
END_METHOD

END_PROGRAM

// ---- POUs/A_Master/PRG_FaultHandling.TcPOU
PROGRAM PRG_FaultHandling
VAR
	
	i							: INT;
	bFlagResetOn				: BOOL;
	bStationCycleFaultFlag		: BOOL;




END_VAR
VAR_IN_OUT

  aAlarms  : ARRAY[0..3] OF ST_Events;
END_VAR

ACT_FaultTrig();

(************************************** Faults reset **********************************************)
IF   GVL_HMI_GLOBAL.bResetButton THEN 
	FOR i := 0 TO 127 DO
		GVL_MASTER.stAlarms[0].aEventFlags[i] := FALSE;
	END_FOR
END_IF


//===============================================================
//Initialize event texts on first scan
IF NOT GVL_MASTER.stAlarms[0].bEventTextsSet THEN
	SetEventTexts();
	GVL_MASTER.stAlarms[0].bEventTextsSet := TRUE;
END_IF
IF NOT GVL_MASTER.stAlarms[0].bEventTextsSet THEN
	GVL_MASTER.stAlarms[0].bEventTextsSet := FALSE;
END_IF


(***************************************************************************************************)
//Immediate fault
GVL_MASTER.stAlarms[0].bImmediateFault := FALSE;
FOR i := 0 TO 32DO
	GVL_MASTER.stAlarms[0].bImmediateFault := GVL_MASTER.stAlarms[0].bImmediateFault OR GVL_MASTER.stAlarms[0].aEventFlags[i];
END_FOR

//Cycle stop fault
GVL_MASTER.stAlarms[0].bCycleStopFault := FALSE;
FOR i := 33 TO 79 DO
	GVL_MASTER.stAlarms[0].bCycleStopFault := GVL_MASTER.stAlarms[0].bCycleStopFault OR GVL_MASTER.stAlarms[0].aEventFlags[i];
END_FOR

//Cycle stop request
GVL_MASTER.stAlarms[0].bCycleStopRequest := FALSE;
FOR i := 80 TO 99 DO
	GVL_MASTER.stAlarms[0].bCycleStopRequest := GVL_MASTER.stAlarms[0].bCycleStopRequest OR GVL_MASTER.stAlarms[0].aEventFlags[i];
END_FOR


(**************************** Master Fault Monitors ***********************************************)
(* Station Immediate Fault Monitor *)
GVL_MASTER.stMasterControl.bNoStationImmediateFault := 	NOT GVL_MASTER.stAlarms[0].bImmediateFault AND NOT GVL_MASTER.stAlarms[1].bImmediateFault AND
                                            			NOT GVL_MASTER.stAlarms[2].bImmediateFault AND NOT GVL_MASTER.stAlarms[3].bImmediateFault;

(**************************************************************************************************)
(**************************** Cycle stop falt  **************************************)
bStationCycleFaultFlag := NOT GVL_MASTER.stAlarms[0].bCycleStopFault AND NOT GVL_MASTER.stAlarms[1].bCycleStopFault AND
                          NOT GVL_MASTER.stAlarms[2].bCycleStopFault AND NOT GVL_MASTER.stAlarms[3].bCycleStopFault;

(**************************** Master Immediate Fault Monitor **************************************)
GVL_MASTER.stMasterControl.bNoMachineImmediateFault := NOT GVL_MASTER.stAlarms[0].bImmediateFault AND NOT GVL_MASTER.stAlarms[1].bImmediateFault AND
                                            NOT GVL_MASTER.stAlarms[2].bImmediateFault AND NOT GVL_MASTER.stAlarms[3].bImmediateFault;

									
(**************************************************************************************************)

(* Master Cycle Stop Fault Monitor *)
GVL_MASTER.stMasterControl.bNoCycleStopFault := NOT GVL_MASTER.stAlarms[0].bCycleStopFault AND NOT GVL_MASTER.stAlarms[1].bCycleStopFault
												AND NOT GVL_MASTER.stAlarms[2].bCycleStopFault AND NOT GVL_MASTER.stAlarms[3].bCycleStopFault;

ACTION ACT_FaultTrig:
 (**************************************************************************************************)
(**************************** Master Immediate Fault Stop *****************************************)
(**************************************************************************************************)

//Beckhoff EL1809 Not Operational
IF NOT GVL_MASTER.stMachineStatus.bSystemPowerUp AND GVL_IO.dwTerminalInfo[3].nTerminal_State<>8 THEN
	GVL_MASTER.stAlarms[0].aEventFlags[33] := TRUE;
END_IF
//Beckhoff EL2809 Not Operational
IF NOT GVL_MASTER.stMachineStatus.bSystemPowerUp AND GVL_IO.dwTerminalInfo[4].nTerminal_State<>8 THEN
	GVL_MASTER.stAlarms[0].aEventFlags[34] := TRUE;
END_IF
//Cognex  IS2801M Connection Erro
IF NOT GVL_MASTER.stMachineStatus.bSystemPowerUp AND GVL_IO.dwBoxInfo[15].nPnIoBoxState<>0 THEN
	GVL_MASTER.stAlarms[0].aEventFlags[35] := TRUE;
END_IF

//Cognex  IS2801M Diagnostic Error
IF NOT GVL_MASTER.stMachineStatus.bSystemPowerUp AND GVL_IO.dwBoxInfo[15].nPnIoBoxDiag=1 THEN
	GVL_MASTER.stAlarms[0].aEventFlags[37] := TRUE;
END_IF
//System stopping timeout
GVL_MASTER.stAlarms[0].aEventTimers[38](IN := ( GVL_MASTER.stMachineStatus.bSystemStopping ), PT := T#20S);
IF GVL_MASTER.stAlarms[0].aEventTimers[38].Q THEN
	GVL_MASTER.stAlarms[0].aEventFlags[38] := TRUE;	
END_IF
//User not Log In
GVL_MASTER.stAlarms[0].aEventTimers[39](IN := (NOT GVL_HMI_GLOBAL.bUserLogedIntSignal), PT := T#40MS);
IF GVL_MASTER.stAlarms[0].aEventTimers[39].Q THEN
	GVL_MASTER.stAlarms[0].aEventFlags[39] := TRUE;	
END_IF
//User LOG-Off Timeout Manual Mode
GVL_MASTER.stAlarms[0].aEventTimers[40](IN:= ((NOT GVL_HMI_GLOBAL.bUserLogedIntSignal) AND GVL_MASTER.stMachineStatus.bManualMode),PT:= T#1S); 
IF GVL_MASTER.stAlarms[0].aEventTimers[40].Q THEN
	GVL_MASTER.stAlarms[0].aEventFlags[40] := TRUE;
END_IF
//Keyence DL-P1 Error
IF GVL_IO.dw_B08_DL_PN1.dldErrorStt THEN
	GVL_MASTER.stAlarms[0].aEventFlags[41] := TRUE;
END_IF
//10 Min Auto cycle stop
IF PRG_MasterCycle.bAutoCycleStop  THEN //
	GVL_MASTER.stAlarms[0].aEventFlags[80] := TRUE;
END_IF
//Autocyle Timeout 
(*GVL_MASTER.stAlarms[0].aEventTimers[42](IN:= GVL_MASTER.stStationSruct[0].bStationInProgress, PT :=T#10M ); 
IF GVL_MASTER.stAlarms[0].aEventTimers[42].Q THEN
	GVL_MASTER.stAlarms[0].aEventFlags[42] := TRUE;
END_IF*)
//Part removed during process
IF GVL_Master.stStationSruct[0].nState > 1000 AND GVL_Master.stStationSruct[0].nState < 2000 AND NOT GVL_IO.dw_T02_EL1809.iPartPresent THEN
	GVL_MASTER.stAlarms[0].aEventFlags[43] := TRUE;
END_IF
//Clamp toggled before requested
IF GVL_Master.stStationSruct[0].nState > 1000 AND GVL_Master.stStationSruct[0].nState <= 1136 AND GVL_IO.dw_T02_EL1809.iCalmpClosed THEN
	GVL_MASTER.stAlarms[0].aEventFlags[44] := TRUE;
END_IF
//Clamp toggled before requested
IF GVL_Master.stStationSruct[0].nState > 1142 AND GVL_Master.stStationSruct[0].nState < 1700 AND NOT GVL_IO.dw_T02_EL1809.iCalmpClosed THEN
	GVL_MASTER.stAlarms[0].aEventFlags[45] := TRUE;
END_IF
//Press Acknowledge
IF GVL_HMI_GLOBAL.bAutocycleFaultDialog THEN
	GVL_MASTER.stAlarms[0].aEventFlags[46] := TRUE;
END_IF


//Remove Nest **LA 17092025
IF GVL_HMI_GLOBAL.bStartButton AND NOT PRG_Mastercycle.biClamp AND PRG_Mastercycle.biPartPresent THEN 
	GVL_MASTER.stAlarms[0].aEventFlags[100] := TRUE;
	ELSIF NOT PRG_Mastercycle.biPartPresent THEN 
		GVL_MASTER.stAlarms[0].aEventFlags[100] := FALSE;
END_IF

//Release Clamp  **LA 17092025
IF GVL_HMI_GLOBAL.bStartButton AND PRG_Mastercycle.biClamp AND NOT PRG_Mastercycle.biPartPresent AND GVL_MASTER.stMachineStatus.bSystemReadyToStart THEN 
	GVL_MASTER.stAlarms[0].aEventFlags[101] := TRUE;
	ELSIF NOT PRG_Mastercycle.biClamp THEN 
		GVL_MASTER.stAlarms[0].aEventFlags[101] := FALSE;
END_IF

//Releas Clamp and Remove Nest  **LA 17092025
IF GVL_HMI_GLOBAL.bStartButton AND PRG_Mastercycle.biClamp AND PRG_Mastercycle.biPartPresent AND GVL_MASTER.stMachineStatus.bSystemReadyToStart THEN
	GVL_MASTER.stAlarms[0].aEventFlags[102] := TRUE;
	ELSIF  NOT PRG_Mastercycle.biClamp AND NOT PRG_Mastercycle.biPartPresent THEN
		GVL_MASTER.stAlarms[0].aEventFlags[102] := FALSE;
END_IF
END_ACTION

METHOD PRIVATE SetEventTexts : BOOL
VAR_INPUT
END_VAR
//Immediate Faults
GVL_MASTER.stAlarms[0].aEventTexts[0] := 'SPARE';
GVL_MASTER.stAlarms[0].aEventTexts[1] := 'SPARE';
GVL_MASTER.stAlarms[0].aEventTexts[2] := 'SPARE';
GVL_MASTER.stAlarms[0].aEventTexts[3] := 'SPARE';
GVL_MASTER.stAlarms[0].aEventTexts[4] := '';
GVL_MASTER.stAlarms[0].aEventTexts[5] := '';
GVL_MASTER.stAlarms[0].aEventTexts[6] := '';
GVL_MASTER.stAlarms[0].aEventTexts[7] := '';
GVL_MASTER.stAlarms[0].aEventTexts[8] := '';
GVL_MASTER.stAlarms[0].aEventTexts[9] := '';
GVL_MASTER.stAlarms[0].aEventTexts[10] := '';
GVL_MASTER.stAlarms[0].aEventTexts[10] := ''; 
GVL_MASTER.stAlarms[0].aEventTexts[11] := '';
GVL_MASTER.stAlarms[0].aEventTexts[12] := '';
GVL_MASTER.stAlarms[0].aEventTexts[13] := '';
GVL_MASTER.stAlarms[0].aEventTexts[14] := '';
GVL_MASTER.stAlarms[0].aEventTexts[15] := '';


//Cycle stop fault

GVL_MASTER.stAlarms[0].aEventTexts[33] := 'Beckhoff EL1809 Not Operational';
GVL_MASTER.stAlarms[0].aEventTexts[34] := 'Beckhoff EL2809 Not Operational';
GVL_MASTER.stAlarms[0].aEventTexts[35] := 'Cognex  IS2801M Connection Error';
GVL_MASTER.stAlarms[0].aEventTexts[36] := 'External Error - Cognex Camera ERROR';
GVL_MASTER.stAlarms[0].aEventTexts[37] := 'Cognex  IS2801M Diagnostic Error';
GVL_MASTER.stAlarms[0].aEventTexts[38] := 'Master - Stopping timeout';
GVL_MASTER.stAlarms[0].aEventTexts[39] := 'User Not Log IN';
GVL_MASTER.stAlarms[0].aEventTexts[40] := 'User Log-Off Timeout Manual Mode'; 
GVL_MASTER.stAlarms[0].aEventTexts[41] := 'Keyence DL-P1 Error';
GVL_MASTER.stAlarms[0].aEventTexts[42] := 'Autocyle Timeou' ;
GVL_MASTER.stAlarms[0].aEventTexts[43] := 'Part removed during cycle';
GVL_MASTER.stAlarms[0].aEventTexts[44] := 'Clamp toggled before requested';
GVL_MASTER.stAlarms[0].aEventTexts[45] := 'Clamp toggled before requested';
GVL_MASTER.stAlarms[0].aEventTexts[46] := 'Press Acknowledge';
GVL_MASTER.stAlarms[0].aEventTexts[47] := '';
GVL_MASTER.stAlarms[0].aEventTexts[48] := '';
GVL_MASTER.stAlarms[0].aEventTexts[59] := '';
GVL_MASTER.stAlarms[0].aEventTexts[50] := '';

//Cycle Stop Requests

GVL_MASTER.stAlarms[0].aEventTexts[80] := 'Machine Cycle Stop 10 Min Not Use Timeout';
GVL_MASTER.stAlarms[0].aEventTexts[81] := '';
GVL_MASTER.stAlarms[0].aEventTexts[82] := '';

GVL_MASTER.stAlarms[0].aEventTexts[84] := '';
GVL_MASTER.stAlarms[0].aEventTexts[85] := '';
GVL_MASTER.stAlarms[0].aEventTexts[86] := '';
GVL_MASTER.stAlarms[0].aEventTexts[87] := ''; 
GVL_MASTER.stAlarms[0].aEventTexts[88] := '';
GVL_MASTER.stAlarms[0].aEventTexts[89] := '';


// Message //**LA 15092025
GVL_MASTER.stAlarms[0].aEventTexts[100] := 'Remove Nest';
GVL_MASTER.stAlarms[0].aEventTexts[101] := 'Release Clamp';
GVL_MASTER.stAlarms[0].aEventTexts[102] := 'Release Clamp and Remove Nest';
END_METHOD

END_PROGRAM

// ---- POUs/A_Master/PRG_MasterCycle.TcPOU
PROGRAM PRG_MasterCycle
VAR
	
		tonCaseTimDelay    	: ARRAY [1..20] OF Tc2_Standard.TON;
	    rtrigCaseTriger    	: ARRAY [1..10] OF Tc2_Standard.R_TRIG;
		ftrigCaseTriger		: ARRAY [1..10] OF Tc2_Standard.F_TRIG;
	   	rtrigFaultMachine  	: Tc2_Standard.R_TRIG;	
		
		biClamp				: BOOL;
		biPartPresent		: BOOL;
		


		bAutoCycleStop		: BOOL;
		
		bCycleFlag			: BOOL;
		bGreenLED			: BOOL;
		bRedLED				: BOOL;
		bEndCycleFlag		: BOOL;
		bStationsStopped	: BOOL;
		bHeighTestCompleteFlag : BOOL;
		bLeakTestCompleteFlag : BOOL;
		i					: DINT;
		
		


END_VAR
VAR_IN_OUT
	stStationStruct          : ST_StandardStationStruct;
END_VAR

ACT_LinkIO();
ACT_TimTrig();
stStationStruct.bStationInProgress := stStationStruct.nState>=1100 AND stStationStruct.nState<=1600;

IF stStationStruct.nState <700 OR  stStationStruct.nState > 4000 THEN
	GVL_HMI_GLOBAL.sActualProcess := ""; 
	GVL_MASTER.stNest.bPiecePass 	:= FALSE;
	GVL_MASTER.stNest.bPieceReject 	:= FALSE;
	bGreenLED						:= FALSE;
	bRedLED							:= FALSE;
	GVL_MASTER.stNest.bHeightPass 	:= FALSE;
	GVL_MASTER.stNest.bVisionPass 	:= FALSE;
	GVL_MASTER.stNest.bHeightReject := FALSE;
	GVL_MASTER.stNest.bVisionReject := FALSE;
END_IF

IF rtrigCaseTriger[3].Q THEN
GVL_PERSIST.stPartsInspection.nPartsGood:= GVL_PERSIST.stPartsInspection.nPartsGood +1;
GVL_PERSIST.stPartsInspection.nTotalPartsGood := GVL_PERSIST.stPartsInspection.nTotalPartsGood+1;
ELSIF GVL_HMI_GLOBAL.bResetGoodParts THEN
GVL_PERSIST.stPartsInspection.nPartsGood:=0;	
END_IF


IF rtrigCaseTriger[4].Q THEN
	GVL_PERSIST.stPartsInspection.nPartsFailed:=GVL_PERSIST.stPartsInspection.nPartsFailed+1;
	GVL_PERSIST.stPartsInspection.nTotalPartsFailed:= GVL_PERSIST.stPartsInspection.nTotalPartsFailed+1;
ELSIF GVL_HMI_GLOBAL.bResetFailedParts THEN
	GVL_PERSIST.stPartsInspection.nPartsFailed:=0;
END_IF

IF stStationStruct.nState < 700 THEN
	 GVL_HMI_GLOBAL.sMessageToOperator := "Press Reset Button to Home Machine";
END_IF

CASE stStationStruct.nState OF
	
100: 
   bAutoCycleStop := FALSE;
IF NOT GVL_MASTER.stMachineStatus.bSystemPowerUp THEN
	stStationStruct.nState := 200;
END_IF
200:
IF GVL_MASTER.stMachineStatus.bSystemInitialising THEN
	stStationStruct.nState := 300;
END_IF
300:
   GVL_Master.stStationSruct[1].bStationInitRequest := TRUE;
   GVL_Master.stStationSruct[3].bStationInitRequest := TRUE;
   
IF GVL_Master.stStationSruct[1].bStationInitRequest AND
   GVL_Master.stStationSruct[3].bStationInitRequest  THEN
	stStationStruct.nState := 400;
END_IF
400:
IF NOT GVL_Master.stStationSruct[1].bStationInitRequest AND
   NOT GVL_Master.stStationSruct[3].bStationInitRequest THEN
	stStationStruct.nState := 500;   
END_IF 
500:
   GVL_Master.stStationSruct[1].bStationAcknowledge := TRUE;
   GVL_Master.stStationSruct[3].bStationAcknowledge := TRUE;
IF   GVL_Master.stStationSruct[1].bStationAcknowledge AND
     GVL_Master.stStationSruct[3].bStationAcknowledge THEN
     stStationStruct.nState := 600;
END_IF
600:
IF GVL_Master.stStationSruct[1].bStationHomed AND GVL_Master.stStationSruct[3].bStationHomed  THEN
   GVL_Master.stStationSruct[1].bStationAcknowledge := FALSE;
   GVL_Master.stStationSruct[3].bStationAcknowledge := FALSE;
   stStationStruct.nState := 700;
END_IF
700: // All Station Homed and waiting for Autocycle 
   bAutoCycleStop := FALSE;
   GVL_HMI_GLOBAL.sActualProcess := "Waiting for Autocycle";
   IF GVL_MASTER.stMachineStatus.bSystemReadyToStart THEN 
	  GVL_HMI_GLOBAL.sMessageToOperator := "Press Start Button to Autocycle";
   ELSE GVL_HMI_GLOBAL.sMessageToOperator := "Press Reset Button to Reset machine";
   END_IF
   
IF GVL_Master.stMachineStatus.bSystemAutoCycle THEN
	stStationStruct.nState := 800;
ELSIF GVL_Master.stMachineStatus.bManualMode THEN
      stStationStruct.nState := 4000;
ELSIF GVL_Master.stMachineStatus.bSystemStopping AND NOT bStationsStopped  THEN
      stStationStruct.nState := 5000;
ELSIF GVL_Master.stMachineStatus.bCycleStopFault OR GVL_Master.stMachineStatus.bImmediateFault THEN
      stStationStruct.nState := 6000;	  
END_IF

IF tonCaseTimDelay[9].Q THEN
	stStationStruct.nState := 1000;
END_IF
800:
stStationStruct.nState := 1000;
1000: // System Autocycle

IF biPartPresent AND bEndCycleFlag THEN
	GVL_HMI_GLOBAL.sMessageToOperator := "Remove Part";
ELSE GVL_HMI_GLOBAL.sMessageToOperator := "Insert Part to begin process";
END_IF


IF  rtrigCaseTriger [5].Q  AND NOT bEndCycleFlag THEN
	GVL_MASTER.stNest.bHeightPass 	:= FALSE;
	GVL_MASTER.stNest.bVisionPass 	:= FALSE;
	GVL_MASTER.stNest.bHeightReject := FALSE;
	GVL_MASTER.stNest.bVisionReject := FALSE;
	GVL_MASTER.stNest.bPiecePass 	:= FALSE;
	GVL_MASTER.stNest.bPieceReject 	:= FALSE;
	GVL_MASTER.stNest.bNestPartProced := FALSE;
	GVL_MASTER.stNest.sHeightHMI 	:= "";
	GVL_MASTER.stNest.sVisionHMI 	:= "";
	GVL_MASTER.stNest.sPieceHMI 	:= "";
	bCycleFlag						:= TRUE;
	GVL_HMI_GLOBAL.sMessageToOperator := "Process in progress";
	GVL_HMI_GLOBAL.bResetPassAndFail:= TRUE;
	GVL_HMI_GLOBAL.sActualProcess := "";
	bGreenLED						:= FALSE;
	bRedLED							:= FALSE;
	GVL_HMI_GLOBAL.bRejectPieceAcknowledge := FALSE;
	stStationStruct.nState 			:= 1130;
	
ELSIF GVL_Master.stMachineStatus.bSystemStopping  THEN
      stStationStruct.nState := 5000;
ELSIF tonCaseTimDelay[10].Q THEN
	  bAutoCycleStop := TRUE;
      stStationStruct.nState := 5000;	
END_IF
1130:
IF tonCaseTimDelay[13].Q THEN
	GVL_HMI_GLOBAL.bResetPassAndFail:= FALSE;
	stStationStruct.nState 			:= 1132;
END_IF


//Vision Test
1132: 
	GVL_MASTER.anValueBeforeMeasurement := GVL_MASTER.aSensorCurrentValue;
	GVL_HMI_GLOBAL.sActualProcess := "Vision process"; 
	GVL_Master.stStationSruct[3].bStationRequest := TRUE;
	stStationStruct.nState := 1134;
1134:
IF GVL_Master.stStationSruct[3].bStationInProgress THEN
	stStationStruct.nState := 1136;
END_IF
1136:
IF GVL_Master.stStationSruct[3].bStationComplete AND NOT GVL_Master.stMachineStatus.bSystemStopping THEN
	stStationStruct.nState := 1138;
ELSIF GVL_Master.stMachineStatus.bSystemStopping OR ftrigCaseTriger [1].Q THEN
	stStationStruct.nState := 5000;
END_IF
1138:
GVL_HMI_GLOBAL.sMessageToOperator := "Toggle Clamp to continue the process";
IF rtrigCaseTriger [1].Q  THEN
	stStationStruct.nState := 1142;
ELSIF GVL_Master.stMachineStatus.bSystemStopping  THEN
      stStationStruct.nState := 5000;
ELSIF tonCaseTimDelay[10].Q THEN
	  bAutoCycleStop := TRUE;
      stStationStruct.nState := 5000;	

END_IF
//Height Test
1142: 
	GVL_HMI_GLOBAL.sMessageToOperator := "Process in progress";
	GVL_HMI_GLOBAL.sActualProcess := "Height test process"; 
	GVL_Master.stStationSruct[1].bStationRequest := TRUE;
	stStationStruct.nState := 1144;
1144:
IF GVL_Master.stStationSruct[1].bStationInProgress THEN
	stStationStruct.nState := 1146;
END_IF
1146:
IF GVL_Master.stStationSruct[1].bStationComplete THEN
		stStationStruct.nState := 1152;
		GVL_MASTER.bHeightTestacknowledge := TRUE;
ELSIF GVL_Master.stMachineStatus.bSystemStopping THEN
	stStationStruct.nState := 5000;
END_IF
1152: 
	GVL_MASTER.stNest.bNestPartProced 	:= TRUE;
	bHeighTestCompleteFlag				:= FALSE;
	bLeakTestCompleteFlag				:= FALSE;
IF tonCaseTimDelay[12].Q THEN
	GVL_MASTER.bHeightTestacknowledge := FALSE;
	stStationStruct.nState := 1220;
END_IF
	
1220:
IF GVL_MASTER.stNest.bHeightPass AND GVL_MASTER.stNest.bVisionPass THEN
	GVL_MASTER.stNest.bPiecePass 	:= TRUE;
	GVL_MASTER.stNest.bPieceReject 	:= FALSE;
	GVL_MASTER.stNest.sPieceHMI 	:= "Pass";
	bGreenLED						:= TRUE;
	bRedLED							:= FALSE;
ELSE GVL_MASTER.stNest.bNestPartOK := FALSE;
	GVL_MASTER.stNest.sPieceHMI 	:= "Fail";
	GVL_MASTER.stNest.bPiecePass 	:= FALSE;
	GVL_MASTER.stNest.bPieceReject 	:= TRUE;
	bGreenLED						:= FALSE;
	bRedLED							:= TRUE;
END_IF
GVL_MASTER.stNest.sDate := GVL_HMI_GLOBAL.sSystemDate;
GVL_MASTER.stNest.sTime := GVL_HMI_GLOBAL.sSystemTime;

IF rtrigCaseTriger [8].Q THEN	
	
	FOR i :=200 TO 2 BY (-1) DO
		GVL_HMI_GLOBAL.aStatistics[i]	:= GVL_HMI_GLOBAL.aStatistics[i-1];
	END_FOR
	
	GVL_HMI_GLOBAL.aStatistics[1] := GVL_MASTER.stNest;
END_IF

IF tonCaseTimDelay[11].Q THEN
	stStationStruct.nState := 1500;
END_IF

1500:
IF GVL_Master.stStationSruct[1].bStationNotMoving  AND GVL_Master.stStationSruct[3].bStationNotMoving THEN
	stStationStruct.nState := 1550;
END_IF
1550:
IF  GVL_MASTER.stNest.bPiecePass THEN	
	stStationStruct.nState := 1600;
ELSIF  GVL_MASTER.stNest.bPieceReject AND GVL_HMI_GLOBAL.bRejectPieceAcknowledge THEN
	stStationStruct.nState := 1600;
END_IF

1600:
GVL_HMI_GLOBAL.sMessageToOperator 				:= "Cycle Complete";   // **LAA 17092025
bEndCycleFlag	:= TRUE;
IF NOT GVL_MASTER.stMachineStatus.bSystemStopping  THEN 
	stStationStruct.nState := 1700;
ELSE 
    stStationStruct.nState := 5000;	
END_IF
1700:
GVL_HMI_GLOBAL.sMessageToOperator 				:= "Release Clamp";    // **LAA 17092025
IF rtrigCaseTriger [7].Q  THEN 
	stStationStruct.nState := 1000; 
END_IF

4000: 
IF NOT GVL_MASTER.stMachineStatus.bManualMode THEN
	stStationStruct.nState := 700;	
ELSIF GVL_MASTER.stMachineStatus.bCycleStopFault OR GVL_MASTER.stMachineStatus.bImmediateFault THEN
      stStationStruct.nState := 6000;		
END_IF

//stopping
5000:
	GVL_Master.stStationSruct[1].bNoCycleStopRequest := FALSE;
	GVL_Master.stStationSruct[3].bNoCycleStopRequest := FALSE;
	

IF tonCaseTimDelay[6].Q AND (GVL_Master.stStationSruct[1].nState = 1000) 
                        AND (GVL_Master.stStationSruct[3].nState < 1100) THEN
	bAutoCycleStop := FALSE;
	
	stStationStruct.nState := 700;

	
END_IF

6000:
IF tonCaseTimDelay[1].Q THEN
	GVL_Master.stStationSruct[1].bStationInitRequest := FALSE;
	GVL_Master.stStationSruct[2].bStationInitRequest := FALSE;
	GVL_Master.stStationSruct[3].bStationInitRequest := FALSE;
	GVL_Master.stStationSruct[1].bStationRequest := FALSE;
	GVL_Master.stStationSruct[2].bStationRequest := FALSE;
    GVL_Master.stStationSruct[3].bStationRequest := FALSE;
	GVL_Master.stStationSruct[1].bStationAbort := TRUE;
    GVL_Master.stStationSruct[2].bStationAbort := TRUE;
	GVL_Master.stStationSruct[3].bStationAbort := TRUE;
	stStationStruct.nState := 100;
END_IF


END_CASE

//++++++++++++++++++++++++++++++++++++++++++++++++++++++++++++++++++++++++++++++++++++++++++++++++++++++++++++++++++++++++++++++++++++++

IF rtrigFaultMachine.Q THEN
   stStationStruct.nState := 6000;	  
END_IF

IF  (stStationStruct.nState = 4000) OR (stStationStruct.nState = 5000) OR (stStationStruct.nState = 6000) THEN
   GVL_Master.stStationSruct[1].bStationAcknowledge := FALSE;
   GVL_Master.stStationSruct[2].bStationAcknowledge := FALSE;
   GVL_Master.stStationSruct[3].bStationAcknowledge := FALSE;
   GVL_Master.stStationSruct[1].bStationInitRequest := FALSE;
   GVL_Master.stStationSruct[2].bStationInitRequest := FALSE;
   GVL_Master.stStationSruct[3].bStationInitRequest := FALSE;
END_IF

ACTION ACT_LinkIO:
// Initialisation Progres
IF GVL_Master.stStationSruct[1].bStationInProgressInit THEN
	GVL_Master.stStationSruct[1].bStationInitRequest := FALSE;
END_IF
IF GVL_Master.stStationSruct[2].bStationInProgressInit THEN
	GVL_Master.stStationSruct[2].bStationInitRequest := FALSE;
END_IF
IF GVL_Master.stStationSruct[3].bStationInProgressInit THEN
	GVL_Master.stStationSruct[3].bStationInitRequest := FALSE;
END_IF

// Cycle Progres
IF GVL_Master.stStationSruct[1].bStationInProgress THEN
	GVL_Master.stStationSruct[1].bStationRequest := FALSE;
END_IF
IF GVL_Master.stStationSruct[2].bStationInProgress THEN
	GVL_Master.stStationSruct[2].bStationRequest := FALSE;
END_IF
IF GVL_Master.stStationSruct[3].bStationInProgress THEN
	GVL_Master.stStationSruct[3].bStationRequest := FALSE;
END_IF

// Abort Station
IF GVL_Master.stStationSruct[1].nState = 100 THEN
	GVL_Master.stStationSruct[1].bStationAbort := FALSE;
END_IF
IF GVL_Master.stStationSruct[2].nState = 100 THEN	
    GVL_Master.stStationSruct[2].bStationAbort := FALSE;
END_IF	
IF GVL_Master.stStationSruct[3].nState = 100 THEN
	GVL_Master.stStationSruct[3].bStationAbort := FALSE;
END_IF

IF (GVL_Master.stStationSruct[1].nState = 100) OR (GVL_Master.stStationSruct[1].nState = 1000) THEN
	GVL_Master.stStationSruct[1].bNoCycleStopRequest := TRUE;
END_IF
IF (GVL_Master.stStationSruct[2].nState = 100) OR (GVL_Master.stStationSruct[2].nState = 1000) THEN	
    GVL_Master.stStationSruct[2].bNoCycleStopRequest := TRUE;
END_IF
IF (GVL_Master.stStationSruct[3].nState = 100) OR (GVL_Master.stStationSruct[3].nState = 1000) THEN	
	GVL_Master.stStationSruct[3].bNoCycleStopRequest := TRUE;
END_IF

IF  (GVL_Master.stStationSruct[1].nState = 1000) AND (GVL_Master.stStationSruct[2].nState = 1000) 
                        AND (GVL_Master.stStationSruct[3].nState = 1000) THEN
	bStationsStopped := TRUE;
ELSE bStationsStopped := FALSE;

END_IF

GVL_MASTER.stMasterControl.bAllStationsCycledStopped := (GVL_Master.stStationSruct[1].nState < 1100)
                                         AND (GVL_Master.stStationSruct[3].nState = 1000)
										 AND  stStationStruct.nState=700;
										 
	biClamp									:= GVL_IO.dw_T02_EL1809.iCalmpClosed;
	biPartPresent							:=  GVL_IO.dw_T02_EL1809.iPartPresent;
	GVL_MASTER.stNest.bNestPresent			:= GVL_IO.dw_T02_EL1809.iCalmpClosed;
	GVL_IO.dw_T03_EL2809.qPassIndicatorGreen:= bGreenLED;
	GVL_IO.dw_T03_EL2809.qRejectIndicatorRed:= bRedLED;
	
IF ftrigCaseTriger[1].Q THEN
	bEndCycleFlag							:= FALSE;
END_IF
	
GVL_MASTER.aSensorCurrentValue[1] 					:= GVL_IO.dw_B08_DL_PN1.gt2_1_1CurrentValue;
GVL_MASTER.aSensorCurrentValue[2] 					:= GVL_IO.dw_B08_DL_PN1.gt2_1_2CurrentValue;
GVL_MASTER.aSensorCurrentValue[3] 					:= GVL_IO.dw_B08_DL_PN1.gt2_1_3CurrentValue;
GVL_MASTER.aSensorCurrentValue[4] 					:= GVL_IO.dw_B08_DL_PN1.gt2_2CurrentValue;
END_ACTION

ACTION ACT_TimTrig:
tonCaseTimDelay[1](IN:= (stStationStruct.nState = 6000),PT:=T#100MS); //
tonCaseTimDelay[2](IN:= (stStationStruct.nState = 5000),PT:=T#100MS); //
tonCaseTimDelay[3](IN:= (stStationStruct.nState = 1100),PT:=T#40MS);  //
tonCaseTimDelay[4](IN:= (stStationStruct.nState = 1140),PT:=T#250MS);
tonCaseTimDelay[5](IN:= (stStationStruct.nState = 1900),PT:=T#250MS);
tonCaseTimDelay[6](IN:= (stStationStruct.nState = 5000),PT:=T#250MS);
tonCaseTimDelay[7](IN:= (stStationStruct.nState = 1340),PT:=T#200MS);
tonCaseTimDelay[8](IN:= (stStationStruct.nState = 1320),PT:=T#500MS);
tonCaseTimDelay[9](IN:= (stStationStruct.nState = 800),PT:=T#3S);
tonCaseTimDelay[10](IN:= (stStationStruct.nState = 1000),PT:=T#10M);
tonCaseTimDelay[11](IN:= (stStationStruct.nState = 1220),PT:=T#1S);
tonCaseTimDelay[12](IN:= stStationStruct.nState = 1152,PT:=T#1S );
tonCaseTimDelay[13](IN:=(stStationStruct.nState = 1130),PT:=T#1S );
tonCaseTimDelay[14](IN:= biPartPresent,PT:=T#2S);
tonCaseTimDelay[15](IN:= );
tonCaseTimDelay[16](IN:= );
tonCaseTimDelay[17](IN:= );
tonCaseTimDelay[18](IN:= );
tonCaseTimDelay[19](IN:= );
tonCaseTimDelay[20](IN:= );

rtrigCaseTriger [1](CLK:= biClamp);
rtrigCaseTriger [2](CLK:= tonCaseTimDelay[2].Q);
rtrigCaseTriger [3](CLK:= GVL_MASTER.stNest.bPiecePass);
rtrigCaseTriger [4](CLK:= GVL_MASTER.stNest.bPieceReject);
rtrigCaseTriger [5](CLK:= tonCaseTimDelay[14].Q );
rtrigCaseTriger [6](CLK:= );
rtrigCaseTriger [7](CLK:= NOT biClamp);  // **LAA 17092025);
rtrigCaseTriger [8](CLK:= stStationStruct.nState = 1220);
rtrigCaseTriger [9](CLK:= );
rtrigCaseTriger [10](CLK:= );
rtrigFaultMachine(CLK:= GVL_MASTER.stMachineStatus.bCycleStopFault OR GVL_MASTER.stMachineStatus.bImmediateFault);

ftrigCaseTriger [1](CLK:= biPartPresent );
END_ACTION

END_PROGRAM

// ---- POUs/D_VisionTest/PRG_Fault_VisionTest.TcPOU
PROGRAM PRG_Fault_VisionTest
VAR
	
			i				: INT;
			
END_VAR
VAR_IN_OUT

  aAlarms  : ARRAY[0..3] OF ST_Events;
END_VAR

ACT_FaultTrig();

(************************************** Faults reset **********************************************)
IF   GVL_HMI_GLOBAL.bResetButton THEN 
	FOR i := 0 TO 127 DO
		GVL_MASTER.stAlarms[3].aEventFlags[i] := FALSE;
	END_FOR
END_IF
//===============================================================
//Initialize event texts on first scan
IF NOT GVL_MASTER.stAlarms[3].bEventTextsSet THEN
	SetEventTexts();
	GVL_MASTER.stAlarms[3].bEventTextsSet := TRUE;
END_IF


(***************************************************************************************************)
//Immediate fault
GVL_MASTER.stAlarms[3].bImmediateFault := FALSE;
FOR i := 0 TO 32DO
	GVL_MASTER.stAlarms[3].bImmediateFault := GVL_MASTER.stAlarms[3].bImmediateFault OR GVL_MASTER.stAlarms[3].aEventFlags[i];
END_FOR

//Cycle stop fault
GVL_MASTER.stAlarms[3].bCycleStopFault := FALSE;
FOR i := 33 TO 79 DO
	GVL_MASTER.stAlarms[3].bCycleStopFault := GVL_MASTER.stAlarms[3].bCycleStopFault OR GVL_MASTER.stAlarms[3].aEventFlags[i];
END_FOR
//Cycle stop Request
GVL_MASTER.stAlarms[3].bCycleStopRequest := FALSE;
FOR i := 80 TO 99 DO
	GVL_MASTER.stAlarms[3].bCycleStopRequest := GVL_MASTER.stAlarms[3].bCycleStopRequest OR GVL_MASTER.stAlarms[3].aEventFlags[i];
END_FOR

ACTION ACT_FaultTrig:
(**************************************************************************************************)
(**************************** Master Immediate Fault Stop *****************************************)
(**************************************************************************************************)
(* Copy Safety Immediate Stop Faults to Master Immediate Stop Faults *)

//Camera Station Cycle Timeout
(*GVL_MASTER.stAlarms[3].aEventTimers[1](IN:= (GVL_Master.stStationSruct[3].nState>=1100 AND GVL_Master.stStationSruct[3].nState<1900) ,PT:=T#5S);
IF GVL_MASTER.stAlarms[3].aEventTimers[1].Q THEN // 
	GVL_MASTER.stAlarms[3].aEventFlags[1] := TRUE;
END_IF*)
//Camera Error
GVL_MASTER.stAlarms[3].aEventTimers[2](IN := (NOT PRG_VisionTest.bCamerraNoError),PT:=T#100MS);
IF GVL_MASTER.stAlarms[3].aEventTimers[2].Q THEN //
	GVL_MASTER.stAlarms[3].aEventFlags[2] := TRUE;
END_IF

//Camera No Running
GVL_MASTER.stAlarms[3].aEventTimers[3](IN := (NOT PRG_VisionTest.bOnline),PT:=T#100MS);
IF GVL_MASTER.stAlarms[3].aEventTimers[3].Q THEN //
	GVL_MASTER.stAlarms[3].aEventFlags[3] := TRUE;
END_IF
END_ACTION

METHOD PRIVATE SetEventTexts : BOOL
VAR_INPUT
END_VAR
//Immediate Faults
GVL_MASTER.stAlarms[3].aEventTexts[0] := '';
GVL_MASTER.stAlarms[3].aEventTexts[1] := 'Camera Station Cycle Timeout';
GVL_MASTER.stAlarms[3].aEventTexts[2] := 'Camera Error';
GVL_MASTER.stAlarms[3].aEventTexts[3] := 'Camera No Running';
GVL_MASTER.stAlarms[3].aEventTexts[4] := '';
GVL_MASTER.stAlarms[3].aEventTexts[5] := '';
GVL_MASTER.stAlarms[3].aEventTexts[6] := '';
GVL_MASTER.stAlarms[3].aEventTexts[7] := '';
GVL_MASTER.stAlarms[3].aEventTexts[8] := '';
GVL_MASTER.stAlarms[3].aEventTexts[9] := ''; 
GVL_MASTER.stAlarms[3].aEventTexts[10] := ''; 
GVL_MASTER.stAlarms[3].aEventTexts[11] := '';
GVL_MASTER.stAlarms[3].aEventTexts[12] := '';
GVL_MASTER.stAlarms[3].aEventTexts[13] := '';
GVL_MASTER.stAlarms[3].aEventTexts[14] := '';
GVL_MASTER.stAlarms[3].aEventTexts[15] := '';
GVL_MASTER.stAlarms[3].aEventTexts[16] := '';
GVL_MASTER.stAlarms[3].aEventTexts[17] := '';
GVL_MASTER.stAlarms[3].aEventTexts[18] := '';
GVL_MASTER.stAlarms[3].aEventTexts[19] := '';
GVL_MASTER.stAlarms[3].aEventTexts[20] := '';
GVL_MASTER.stAlarms[3].aEventTexts[21] := '';
GVL_MASTER.stAlarms[3].aEventTexts[22] := '';
GVL_MASTER.stAlarms[3].aEventTexts[28] := '';
GVL_MASTER.stAlarms[3].aEventTexts[29] := '';
GVL_MASTER.stAlarms[3].aEventTexts[30] := '';

//Cycle Stop Requests

GVL_MASTER.stAlarms[3].aEventTexts[80] := '';
GVL_MASTER.stAlarms[3].aEventTexts[81] := '';
GVL_MASTER.stAlarms[3].aEventTexts[82] := '';

GVL_MASTER.stAlarms[3].aEventTexts[84] := '';
GVL_MASTER.stAlarms[3].aEventTexts[85] := '';
GVL_MASTER.stAlarms[3].aEventTexts[86] := '';
GVL_MASTER.stAlarms[3].aEventTexts[87] := ''; 
GVL_MASTER.stAlarms[3].aEventTexts[88] := '';
GVL_MASTER.stAlarms[3].aEventTexts[89] := '';

//Master Messages

GVL_MASTER.stAlarms[3].aEventTexts[100] := '';
GVL_MASTER.stAlarms[3].aEventTexts[101] := '';
GVL_MASTER.stAlarms[3].aEventTexts[102] := '';
GVL_MASTER.stAlarms[3].aEventTexts[103] := '';
GVL_MASTER.stAlarms[3].aEventTexts[104] := '';
GVL_MASTER.stAlarms[3].aEventTexts[105] := '';
GVL_MASTER.stAlarms[3].aEventTexts[106] := '';
END_METHOD

END_PROGRAM

// ---- POUs/D_VisionTest/PRG_VisionTest.TcPOU
PROGRAM PRG_VisionTest
VAR

	biClamp				: BOOL;

	bCamerraNoError     : BOOL;
	bCameraBufOverR     : BOOL;
	bInspectionCompleted: RS;
	bResultValid        : BOOL;
	bJobPass            : BOOL;
	bAqusError          : BOOL;
	bExposComplete      : BOOL;
	bAqusTriggerReady   : BOOL;
	bOnline             : BOOL;
	bTriggerCam         : BOOL;
	bClearBuffer         : BOOL;
	bResetCam      		: BOOL;
	bAcnwResult         : BOOL;
		
	TonCaseDelay  		: ARRAY[1..10] OF Tc2_Standard.TON;
	rtrigCaseTriger  	: ARRAY [1..10] OF Tc2_Standard.R_TRIG;


	nConsParts			: INT;
END_VAR

VAR_IN_OUT
	stStationStruct     : ST_StandardStationStruct;
END_VAR

ACT_IOLink();
ACT_TimTrig();

(************** Station in Home Position **************************)
stStationStruct.bStationHomed :=  (stStationStruct.nState = 1000);

(******************************************************************)
stStationStruct.bStationComplete := stStationStruct.nState = 1900;
stStationStruct.bStationHomingRequest := stStationStruct.nState = 200;
stStationStruct.bStationWaitOnRequest := stStationStruct.nState = 1000; 
stStationStruct.bStationInitDone := stStationStruct.nState = 900;
stStationStruct.bStationInProgressInit := stStationStruct.nState >= 200 AND stStationStruct.nState <= 900;
stStationStruct.bStationInProgress :=  stStationStruct.nState > 1000 AND stStationStruct.nState < 1900;
stStationStruct.bStationWaitOnInit := stStationStruct.nState = 100; 
//stStationStruct.bStationAcknowledge := stStationStruct.nState = 200 OR stStationStruct.nState = 1100;
stStationStruct.bStationNotMoving := stStationStruct.nState = 100 OR stStationStruct.nState = 1000 OR stStationStruct.nState = 1900;
(******************************************************************)
(***************** Counter *************)
IF rtrigCaseTriger[3].Q THEN
GVL_PERSIST.stPartsInspection.nVisionPartsGood:= GVL_PERSIST.stPartsInspection.nVisionPartsGood +1;
GVL_PERSIST.stPartsInspection.nVisionTotalPartsGood := GVL_PERSIST.stPartsInspection.nVisionTotalPartsGood+1;
ELSIF GVL_HMI_GLOBAL.bResetVisionGoodParts THEN
GVL_PERSIST.stPartsInspection.nVisionPartsGood:=0;	
END_IF


IF rtrigCaseTriger[4].Q THEN
	GVL_PERSIST.stPartsInspection.nVisionPartsFailed:=GVL_PERSIST.stPartsInspection.nVisionPartsFailed+1;
	GVL_PERSIST.stPartsInspection.nVisionTotalPartsFailed:= GVL_PERSIST.stPartsInspection.nVisionTotalPartsFailed+1;
ELSIF GVL_HMI_GLOBAL.bResetVisionBadParts THEN
	GVL_PERSIST.stPartsInspection.nVisionPartsFailed:=0;
END_IF

IF rtrigCaseTriger[4].Q THEN
	nConsParts:= nConsParts+1;
ELSIF rtrigCaseTriger[3].Q OR GVL_HMI_GLOBAL.bResetButton THEN
    nConsParts:=0;	
END_IF

bClearBuffer := GVL_HMI_GLOBAL.bResetButton;

(***************************************)

IF rtrigCaseTriger[5].Q THEN
	stStationStruct.nState := 100;
END_IF

(***************************************)


CASE stStationStruct.nState OF
100: 
IF stStationStruct.bStationInitRequest THEN
	 stStationStruct.nState := 140;
END_IF
140:
bClearBuffer := TRUE;
IF bClearBuffer THEN
	stStationStruct.nState := 160;
END_IF
160:
IF tonCaseDelay[8].Q THEN
	bClearBuffer := FALSE;
	stStationStruct.nState := 200;
END_IF
200: // Check if error 
IF bCamerraNoError THEN
	 stStationStruct.nState := 400;
END_IF

400:
IF stStationStruct.bStationAcknowledge THEN
	stStationStruct.nState := 1000;
END_IF
1000: // Waiting for request 

bTriggerCam    := FALSE;

bAcnwResult := FALSE;
bClearBuffer:= FALSE;
IF GVL_HMI_GLOBAL.bResetPassAndFail THEN
	GVL_MASTER.stNest.bVisionPass := FALSE;
	GVL_MASTER.stNest.sVisionHMI := "";
	GVL_MASTER.stNest.bVisionReject := FALSE;
END_IF
IF stStationStruct.bStationRequest AND stStationStruct.bNoCycleStopRequest THEN
   stStationStruct.nState := 1100;  
ELSIF (stStationStruct.bStationManualRequestHMI OR GVL_MASTER.bManualModeTrigger) AND stStationStruct.bNoCycleStopRequest THEN
   stStationStruct.nState := 4000; // Manual Mode
ELSIF stStationStruct.bStationAbort THEN
	   stStationStruct.nState := 100;	   
END_IF
1100:
bTriggerCam := TRUE;
IF bResultValid THEN
	bTriggerCam := FALSE;
	stStationStruct.nState := 1260;
END_IF
1260:// Check Aqusition
IF bInspectionCompleted.Q1 THEN
	stStationStruct.nState := 1270;
END_IF
1270:
IF tonCaseDelay[9].Q THEN
	stStationStruct.nState := 1280;
END_IF

1280: // JOB PASS / JOB FAIL
IF bJobPass  THEN
//   nPartStatus := 1;
	GVL_MASTER.stNest.bVisionPass 	:= TRUE;
	GVL_MASTER.stNest.sVisionHMI 	:= "Pass";
   stStationStruct.nState := 1282;
ELSIF NOT bJobPass  THEN
	//Added checks here not initial for bNestFail or bNestPartReject	
//   nPartStatus := 0;
   GVL_MASTER.stNest.bVisionReject := TRUE;
   GVL_MASTER.stNest.sVisionHMI 	:= "Fail";
   stStationStruct.nState := 1282;
END_IF
1282:
bAcnwResult := TRUE;
bClearBuffer:= TRUE;
IF NOT bResultValid THEN
	stStationStruct.nState := 1284;
END_IF
1284:
bAcnwResult := FALSE;
stStationStruct.nState := 1286;
1286:
IF tonCaseDelay[4].Q THEN
	stStationStruct.nState := 1290;
END_IF

1290:
bTriggerCam    := FALSE;
bAcnwResult 	:= FALSE;
bClearBuffer	:= FALSE;
stStationStruct.nState := 1900;
1900:
IF tonCaseDelay[2].Q AND rtrigCaseTriger[7].Q THEN
	stStationStruct.nState := 1000;
ELSIF NOT stStationStruct.bNoCycleStopRequest AND tonCaseDelay[2].Q THEN
	stStationStruct.nState := 1000;
END_IF
//=== Manual Mode ===
4000:
IF NOT stStationStruct.bStationManualRequestHMI THEN
	stStationStruct.nState := 1000;
END_IF

END_CASE

ACTION ACT_IOLink:

bCamerraNoError      := NOT GVL_IO.dw_B06_KeyenceCamera.bError;
bCameraBufOverR      := GVL_IO.dw_B06_KeyenceCamera.bBusy;
bResultValid		 := GVL_IO.dw_B06_KeyenceCamera.bResultReady;
bInspectionCompleted(SET := GVL_IO.dw_B06_KeyenceCamera.bResultReady, RESET1 := stStationStruct.nState > 1260);

bJobPass             := GVL_IO.dw_B06_KeyenceCamera.bTotalResult;
bAqusError           := GVL_IO.dw_B06_KeyenceCamera.bTriggerFail;
bOnline              := GVL_IO.dw_B06_KeyenceCamera.bRun;


GVL_IO.dw_B06_KeyenceCamera.bTrigger                	:= bTriggerCam;
GVL_IO.dw_B06_KeyenceCamera.bClearBuffer       			:= bClearBuffer;
GVL_IO.dw_B06_KeyenceCamera.bReset                  	:= bResetCam;//--
GVL_IO.dw_B06_KeyenceCamera.bResultReadyAck  			:= bAcnwResult ;

biClamp					:= GVL_IO.dw_T02_EL1809.iCalmpClosed;
END_ACTION

ACTION ACT_TimTrig:
tonCaseDelay[1](IN:= (stStationStruct.nState=400),PT:=T#50MS);
tonCaseDelay[2](IN:= (stStationStruct.nState=1900),PT:=T#100MS);
tonCaseDelay[3](IN:= (stStationStruct.nState=1),PT:=T#100MS);
tonCaseDelay[4](IN:= stStationStruct.nState=1286,PT:=T#500MS);
tonCaseDelay[5](IN:= (stStationStruct.nState=9100),PT:=T#250MS);
tonCaseDelay[6](IN:= (stStationStruct.nState=9200),PT:=T#250MS);
tonCaseDelay[7](IN:= (stStationStruct.nState=1292),PT:=T#50MS);
tonCaseDelay[8](IN:= (stStationStruct.nState=160),PT:=T#250MS);
tonCaseDelay[9](IN:=stStationStruct.nState=1270 ,PT:=T#1S);
tonCaseDelay[10](IN:= ,PT:=T#250MS);

rtrigCaseTriger[1](clk:= stStationStruct.nState>1100);
rtrigCaseTriger[2](clk:= );
rtrigCaseTriger[3](clk:= (stStationStruct.nState=1280) AND bJobPass );
rtrigCaseTriger[4](clk:= (stStationStruct.nState=1280) AND NOT bJobPass );
rtrigCaseTriger[5](clk:= stStationStruct.bStationAbort);
rtrigCaseTriger[6](clk:= (stStationStruct.nState=1240) AND  bAqusError );
rtrigCaseTriger[7](clk:= biClamp);
rtrigCaseTriger[8](clk:= );
rtrigCaseTriger[9](clk:= );
rtrigCaseTriger[10](clk:= );
END_ACTION

END_PROGRAM

// ---- POUs/E_HMI/PRG_HMI.TcPOU
PROGRAM PRG_HMI
VAR
	

	tonCaseDelay				: ARRAY [1..20] OF TON;
	tofCase						: ARRAY [1..20] OF TOF;
	rtrigCaseTriger				: ARRAY [1..20] OF R_TRIG;

	tonResetStatistics			: TON;
END_VAR

ACT_ScreensNamesSet();
ACT_Buttons();
ACT_TimTrig();
ACT_General();

tonResetStatistics( IN := 	GVL_HMI_GLOBAL.aResetHeightSensorBadParts [1] 	OR
							GVL_HMI_GLOBAL.aResetHeightSensorBadParts [2] 	OR
							GVL_HMI_GLOBAL.aResetHeightSensorBadParts [3] 	OR
							GVL_HMI_GLOBAL.aResetHeightSensorBadParts [4] 	OR
							GVL_HMI_GLOBAL.aResetHeightSensorGoodParts[1]	OR
							GVL_HMI_GLOBAL.aResetHeightSensorGoodParts[2]	OR
							GVL_HMI_GLOBAL.aResetHeightSensorGoodParts[3]	OR
							GVL_HMI_GLOBAL.aResetHeightSensorGoodParts[4]	OR
							GVL_HMI_GLOBAL.bResetHeightFailParts			OR
							GVL_HMI_GLOBAL.bResetHeightGoodParts			OR
							GVL_HMI_GLOBAL.bResetGoodParts					OR
							GVL_HMI_GLOBAL.bResetVisionBadParts				OR
							GVL_HMI_GLOBAL.bResetVisionGoodParts			OR
							GVL_HMI_GLOBAL.bResetFailedParts				OR
							GVL_HMI_GLOBAL.bResetGoodParts					,
							PT												:= T#500MS);

ACTION ACT_Buttons:
ACT_TimTrig();

IF tonCaseDelay[1].Q THEN
	
		GVL_HMI_GLOBAL.bResetButton	:= FALSE;
		
END_IF
IF tonCaseDelay[2].Q THEN
	
		GVL_HMI_GLOBAL.bStopButton	:= FALSE;
		
END_IF
IF tonCaseDelay[3].Q THEN
	
		GVL_HMI_GLOBAL.bStartButton	:= FALSE;
		
END_IF



IF tonCaseDelay[7].Q THEN
	
		GVL_HMI_GLOBAL.bShutDown	:= FALSE;
		
END_IF


IF tonCaseDelay[9].Q THEN
	
		GVL_HMI_GLOBAL.bSetSetPointsHeightTest	:= FALSE;
		
END_IF

IF tonCaseDelay[10].Q THEN
	
		GVL_HMI_GLOBAL.bManualMeasureHeightTest	:= FALSE;
		
END_IF

IF tonResetStatistics.Q THEN
	
							GVL_HMI_GLOBAL.aResetHeightSensorBadParts [1] 	:= FALSE;
							GVL_HMI_GLOBAL.aResetHeightSensorBadParts [2] 	:= FALSE;
							GVL_HMI_GLOBAL.aResetHeightSensorBadParts [3] 	:= FALSE;
							GVL_HMI_GLOBAL.aResetHeightSensorBadParts [4] 	:= FALSE;
							GVL_HMI_GLOBAL.aResetHeightSensorGoodParts[1]	:= FALSE;
							GVL_HMI_GLOBAL.aResetHeightSensorGoodParts[2]	:= FALSE;
							GVL_HMI_GLOBAL.aResetHeightSensorGoodParts[3]	:= FALSE;
							GVL_HMI_GLOBAL.aResetHeightSensorGoodParts[4]	:= FALSE;
							GVL_HMI_GLOBAL.bResetHeightFailParts			:= FALSE;
							GVL_HMI_GLOBAL.bResetHeightGoodParts			:= FALSE;
							GVL_HMI_GLOBAL.bResetGoodParts					:= FALSE;
							GVL_HMI_GLOBAL.bResetVisionBadParts				:= FALSE;
							GVL_HMI_GLOBAL.bResetVisionGoodParts			:= FALSE;
							GVL_HMI_GLOBAL.bResetFailedParts				:= FALSE;
							GVL_HMI_GLOBAL.bResetGoodParts					:= FALSE;


END_IF
END_ACTION

ACTION ACT_General:
IF tofCase[1].Q AND 
( NOT GVL_MASTER.stMasterControl.bNoStationImmediateFault OR NOT GVL_MASTER.stMasterControl.bNoCycleStopFault) THEN
	GVL_HMI_GLOBAL.bAutocycleFaultDialog := TRUE;
END_IF
END_ACTION

ACTION ACT_ScreensNamesSet:
GVL_HMI_GLOBAL.aIOScreen[0] := 'Overview';
GVL_HMI_GLOBAL.aIOScreen[1] := 'HMI - CP2913-0000 | Beckhoff HMI';
GVL_HMI_GLOBAL.aIOScreen[2] := 'PLC - C6015-0010 | Beckhoff PLC | Windows 10 Embedded';
GVL_HMI_GLOBAL.aIOScreen[3] := 'Terminal 1- EK1100 | EtherCAT Coupler';
GVL_HMI_GLOBAL.aIOScreen[4] := 'Terminal 2 - EL6070 | Licence ';
GVL_HMI_GLOBAL.aIOScreen[5] := CONCAT('Terminal 3 - ' , GVL_IO.dw_T02_EL1809.sTerminalName);
GVL_HMI_GLOBAL.aIOScreen[6] := CONCAT('Terminal 4 - ' , GVL_IO.dw_T03_EL2809.sTerminalName);
GVL_HMI_GLOBAL.aIOScreen[7] := 'Terminal 12 - EL6631 |  2-port communication interface';
GVL_HMI_GLOBAL.aIOScreen[8] := 'DL-PN1 4Keyence Communication Unit | IV4 Camera | ProfiNET';


GVL_HMI_GLOBAL.aManualScreen[0] := 'Keyence | Vision Test';
GVL_HMI_GLOBAL.aManualScreen[1] := 'Keyence | Height Test';
END_ACTION

ACTION ACT_TimTrig:


tonCaseDelay[1](IN:= GVL_HMI_GLOBAL.bResetButton,PT:=T#500MS);
tonCaseDelay[2](IN:= GVL_HMI_GLOBAL.bStopButton,PT:=T#500MS);
tonCaseDelay[3](IN:= GVL_HMI_GLOBAL.bStartButton,PT:=T#500MS);
tonCaseDelay[4](IN:= ,PT:=T#500MS);
tonCaseDelay[5](IN:= ,PT:=T#500MS);
tonCaseDelay[6](IN:= ,PT:=T#500MS);
//tonCaseDelay[7](IN:= GVL_HMI_GLOBAL.bShutDown,PT:=T#500MS);
tonCaseDelay[8](IN:= ,PT:=T#5S);
tonCaseDelay[9](IN:= GVL_HMI_GLOBAL.bSetSetPointsHeightTest,PT:=T#1S);
tonCaseDelay[10](IN:= GVL_HMI_GLOBAL.bManualMeasureHeightTest,PT:=T#1S);

tofCase[1](IN:= (GVL_Master.stStationSruct[0].nState > 1000 AND GVL_Master.stStationSruct[0].nState < 1900),PT:=T#1S);


rtrigCaseTriger[1](CLK := GVL_MASTER.stNest.bPieceReject);
END_ACTION

END_PROGRAM

// ---- POUs/B_HightTest/PRG_HeightTest.TcPOU
PROGRAM PRG_HeightTest
VAR
	//FUNCTION
	fbHeightMeasurement2						: FB_HeightMeasurement2;
	
	
	bEnable										: BOOL;
	bEnableo									: BOOL;
	bMeasurementRequest							: BOOL;
	bSet										: BOOL;
	bAcknowledge								: BOOL;
	bManualMode									: BOOL;
	bBusy										: BOOL;
	bComplete									: BOOL;

//TrigTim

	rtrigCaseTriger			: ARRAY[1..20] OF R_TRIG;
	tonCaseDelay			: ARRAY[1..10] OF TON;

	
	
END_VAR


VAR_IN_OUT
	stStationStruct          	: ST_StandardStationStruct;
	
END_VAR
VAR PERSISTENT
stHeightMeasurement2						: ST_HeightMeasurement2;
END_VAR

ACT_IOLink();
ACT_TimTrig();
ACT_Statistics();
ACT_ProbesPosition();

(************** Station in Home Position **************************)
stStationStruct.bStationHomed :=  (stStationStruct.nState = 1000);

(******************************************************************)
stStationStruct.bStationComplete := stStationStruct.nState = 1220;
stStationStruct.bStationHomingRequest := stStationStruct.nState = 200;
stStationStruct.bStationWaitOnRequest := stStationStruct.nState = 1000; 
stStationStruct.bStationInitDone := stStationStruct.nState = 400;
stStationStruct.bStationInProgressInit := stStationStruct.nState >= 200 AND stStationStruct.nState <= 900;
stStationStruct.bStationInProgress :=  stStationStruct.nState > 1000 AND stStationStruct.nState < 1900;
stStationStruct.bStationWaitOnInit := stStationStruct.nState = 100; 
//stStationStruct.bStationAcknowledge := stStationStruct.nState = 200 OR stStationStruct.nState = 1100;
stStationStruct.bStationNotMoving := stStationStruct.nState = 100 OR stStationStruct.nState = 1000 OR stStationStruct.nState = 1240;
(******************************************************************)
(***************** Counter *************)


(***************************************)

IF rtrigCaseTriger[5].Q THEN
	stStationStruct.nState := 100;
END_IF

(***************************************)


CASE stStationStruct.nState OF
100:
bMeasurementRequest := FALSE;
IF stStationStruct.bStationInitRequest THEN
	stStationStruct.nState:= 300;
END_IF

300:
IF tonCaseDelay[1].Q THEN
   stStationStruct.nState:= 400;	
END_IF
400:
	stStationStruct.nState:= 1000;

//============== Homed ========================================================

1000:

IF GVL_HMI_GLOBAL.bResetPassAndFail THEN
	bEnable 			:= FALSE;
	bAcknowledge 		:= FALSE;
	bMeasurementRequest	:= FALSE;
	GVL_MASTER.stNest.bHeightPass := FALSE;
	GVL_MASTER.stNest.sHeightHMI := "";
	GVL_MASTER.stNest.bHeightReject := FALSE;

END_IF
IF stStationStruct.bStationRequest AND stStationStruct.bNoCycleStopRequest THEN
   	stStationStruct.nState := 1010;  
ELSIF (stStationStruct.bStationManualRequestHMI OR GVL_MASTER.bManualModeTrigger) AND stStationStruct.bNoCycleStopRequest THEN
   stStationStruct.nState := 4000; // Manual Mode
ELSIF stStationStruct.bStationAbort THEN
	   stStationStruct.nState := 100;	   
END_IF
1010:
bEnable := TRUE;
IF tonCaseDelay[2].Q THEN
	stStationStruct.nState:= 1100;
END_IF
1100:
IF bEnableo THEN
	stStationStruct.nState:= 1110;
END_IF
1110:
bMeasurementRequest := TRUE;
IF NOT bBusy AND bComplete THEN
	bMeasurementRequest := FALSE;
	bAcknowledge		:= TRUE;
	stStationStruct.nState:= 1120;
END_IF
1120: // JOB PASS / JOB FAIL
bAcknowledge			:= FALSE;

IF bComplete AND NOT bBusy  THEN
	GVL_MASTER.stNest.bHeightPass := GVL_HMI_GLOBAL.aGeneralPassHeightTest[5];
	GVL_MASTER.stNest.bHeightReject := GVL_HMI_GLOBAL.aGeneralFailHeightTest[5];
	
	IF GVL_MASTER.stNest.bHeightPass THEN
		GVL_MASTER.stNest.sHeightHMI 	:= "Pass";
		GVL_MASTER.stNest.bHeightPass := TRUE;
		GVL_MASTER.stNest.bHeightReject := FALSE;
	ELSIF  GVL_MASTER.stNest.bHeightReject THEN
		
		GVL_MASTER.stNest.sHeightHMI 	:= "Fail";
		GVL_MASTER.stNest.bHeightPass := FALSE;
		GVL_MASTER.stNest.bHeightReject := TRUE;
	END_IF
	
	stStationStruct.nState:= 1220;
END_IF
1220:

IF tonCaseDelay[5].Q THEN
	stStationStruct.nState:= 1240;
END_IF

1240:
IF (tonCaseDelay[3].Q AND NOT stStationStruct.bStationManualRequestHMI OR GVL_MASTER.bHeightTestacknowledge) OR NOT stStationStruct.bNoCycleStopRequest THEN
	stStationStruct.nState:= 1000;
ELSIF tonCaseDelay[3].Q AND stStationStruct.bStationManualRequestHMI AND stStationStruct.bNoCycleStopRequest THEN
	stStationStruct.nState:= 4000;
END_IF


4000:
IF NOT stStationStruct.bStationManualRequestHMI AND NOT GVL_MASTER.bManualModeTrigger THEN
	stStationStruct.nState := 1000;
	bEnable				:= FALSE;
	bManualMode			:= FALSE;
ELSIF stStationStruct.bStationAbort THEN
	 stStationStruct.nState := 100;
	 bEnable				:= FALSE;
	bManualMode			:= FALSE;
ELSE 
bManualMode			:= TRUE;
bEnable				:= TRUE;	
END_IF



END_CASE

ACTION ACT_IOLink:

stHeightMeasurement2.aSensorCurrentValue[1]		:= DINT_TO_REAL(GVL_IO.dw_B08_DL_PN1.gt2_1_1CurrentValue);
stHeightMeasurement2.aSensorCurrentValue[2]		:= DINT_TO_REAL(GVL_IO.dw_B08_DL_PN1.gt2_1_2CurrentValue);
stHeightMeasurement2.aSensorCurrentValue[3]		:= DINT_TO_REAL(GVL_IO.dw_B08_DL_PN1.gt2_1_3CurrentValue);
stHeightMeasurement2.aSensorCurrentValue[4]		:= DINT_TO_REAL(GVL_IO.dw_B08_DL_PN1.gt2_2CurrentValue);

fbHeightMeasurement2(
	
	aSensorCurrentValue							:= stHeightMeasurement2.aSensorCurrentValue,	
	bEnable										:= bEnable,
	bMeasurementRequest							:= bMeasurementRequest,
	bSetFixedPoints								:= GVL_HMI_GLOBAL.bSetSetPointsHeightTest,
	aTolerance									:= stHeightMeasurement2.aTolerance,
	bAcknowledge								:= bAcknowledge,
	nDistanceBetweenPoints						:= stHeightMeasurement2.nDistanceBetweenPoints,
	anDistanceSetPoint							:= stHeightMeasurement2.anDistanceSetPoint,
	bManualMode									:= bManualMode,
	
	//OUTPUTS
	bBusy										=> bBusy,
	bComplete									=> bComplete,
	bEnableo									=> bEnableo,
	aPass										=> GVL_HMI_GLOBAL.aGeneralPassHeightTest ,
	aFail										=> GVL_HMI_GLOBAL.aGeneralFailHeightTest ,
	aMinLimitCalibrationBlock					=> stHeightMeasurement2.aMinLimitCalibrationBlock,
	aMaxLimitCalibrationBlock					=> stHeightMeasurement2.aMaxLimitCalibrationBlock,
	aDistanceBetweenProbes						=> stHeightMeasurement2.aDistanceBetweenProbes,
	abSensorStuck								=> stHeightMeasurement2.abSensorStuck,
	nFixedPoint									=> stHeightMeasurement2.nFixedPoint,
	aScaledSensorCurrentValue					=> stHeightMeasurement2.aScaledSensorCurrentValue,
	nHeightMeasureStateValue					=> GVL_HMI_GLOBAL.nHeightMeasureStateValue);


//to save data 
GVL_MASTER.stNest.nDistance							:= stHeightMeasurement2.aDistanceBetweenProbes;
GVL_MASTER.stNest.nTarget							:= stHeightMeasurement2.anDistanceSetPoint;
END_ACTION

ACTION ACT_ProbesPosition:
IF ((stHeightMeasurement2.aScaledSensorCurrentValue[1]> GVL_PERSIST.stHeightLimits.nLow)  AND 
	(stHeightMeasurement2.aScaledSensorCurrentValue[1]< GVL_PERSIST.stHeightLimits.nHigh)) AND	
   ((stHeightMeasurement2.aScaledSensorCurrentValue[2]> GVL_PERSIST.stHeightLimits.nLow)  AND 
	(stHeightMeasurement2.aScaledSensorCurrentValue[2]< GVL_PERSIST.stHeightLimits.nHigh)) AND
   ((stHeightMeasurement2.aScaledSensorCurrentValue[3]> GVL_PERSIST.stHeightLimits.nLow)  AND 
	(stHeightMeasurement2.aScaledSensorCurrentValue[3]< GVL_PERSIST.stHeightLimits.nHigh)) AND
   ((stHeightMeasurement2.aScaledSensorCurrentValue[4]> GVL_PERSIST.stHeightLimits.nLow)  AND 
	(stHeightMeasurement2.aScaledSensorCurrentValue[4]< GVL_PERSIST.stHeightLimits.nHigh)) THEN

		GVL_HMI_GLOBAL.bProbesPositionOk				:= TRUE;
ELSE 	GVL_HMI_GLOBAL.bProbesPositionOk				:= FALSE;		
	
END_IF
END_ACTION

ACTION ACT_Statistics:

//GENERAL
IF rtrigCaseTriger[3].Q THEN
GVL_PERSIST.stPartsInspection.nHeightPartsGood:= GVL_PERSIST.stPartsInspection.nHeightPartsGood +1;
GVL_PERSIST.stPartsInspection.nHeightTotalPartsGood := GVL_PERSIST.stPartsInspection.nHeightTotalPartsGood+1;
ELSIF GVL_HMI_GLOBAL.bResetHeightGoodParts THEN
GVL_PERSIST.stPartsInspection.nHeightPartsGood:=0;	
END_IF


IF rtrigCaseTriger[4].Q THEN
	GVL_PERSIST.stPartsInspection.nHeightPartsFailed:=GVL_PERSIST.stPartsInspection.nHeightPartsFailed + 1;
	GVL_PERSIST.stPartsInspection.nHeightTotalPartsFailed:= GVL_PERSIST.stPartsInspection.nHeightTotalPartsFailed + 1;
ELSIF GVL_HMI_GLOBAL.bResetHeightFailParts THEN
	GVL_PERSIST.stPartsInspection.nHeightPartsFailed:=0;
END_IF


//Distance 1

IF rtrigCaseTriger[6].Q THEN
GVL_PERSIST.stPartsInspection.nHeightDistancePartsGood[1]:= GVL_PERSIST.stPartsInspection.nHeightDistancePartsGood[1] +1;
GVL_PERSIST.stPartsInspection.nHeightDistanceTotalPartsGood[1] := GVL_PERSIST.stPartsInspection.nHeightDistanceTotalPartsGood[1]+1;
ELSIF GVL_HMI_GLOBAL.aResetHeightSensorGoodParts[1] THEN
GVL_PERSIST.stPartsInspection.nHeightDistancePartsGood[1]:=0;	
END_IF


IF rtrigCaseTriger[7].Q THEN
	GVL_PERSIST.stPartsInspection.nHeightDistancePartsFailed[1]:=GVL_PERSIST.stPartsInspection.nHeightDistancePartsFailed[1] + 1;
	GVL_PERSIST.stPartsInspection.nHeightDistanceTotalPartsFailed[1]:= GVL_PERSIST.stPartsInspection.nHeightDistanceTotalPartsFailed[1] + 1;
ELSIF GVL_HMI_GLOBAL.aResetHeightSensorBadParts[1] THEN
	GVL_PERSIST.stPartsInspection.nHeightDistancePartsFailed[1]:=0;
END_IF

//Distance 2

IF rtrigCaseTriger[8].Q THEN
GVL_PERSIST.stPartsInspection.nHeightDistancePartsGood[2]:= GVL_PERSIST.stPartsInspection.nHeightDistancePartsGood[2] +1;
GVL_PERSIST.stPartsInspection.nHeightDistanceTotalPartsGood[2] := GVL_PERSIST.stPartsInspection.nHeightDistanceTotalPartsGood[2]+1;
ELSIF GVL_HMI_GLOBAL.aResetHeightSensorGoodParts[2] THEN
GVL_PERSIST.stPartsInspection.nHeightDistancePartsGood[2]:=0;	
END_IF


IF rtrigCaseTriger[9].Q THEN
	GVL_PERSIST.stPartsInspection.nHeightDistancePartsFailed[2]:=GVL_PERSIST.stPartsInspection.nHeightDistancePartsFailed[2] + 1;
	GVL_PERSIST.stPartsInspection.nHeightDistanceTotalPartsFailed[2]:= GVL_PERSIST.stPartsInspection.nHeightDistanceTotalPartsFailed[2] + 1;
ELSIF GVL_HMI_GLOBAL.aResetHeightSensorBadParts[2] THEN
	GVL_PERSIST.stPartsInspection.nHeightDistancePartsFailed[2]:=0;
END_IF

//Distance 3

IF rtrigCaseTriger[10].Q THEN
GVL_PERSIST.stPartsInspection.nHeightDistancePartsGood[3]:= GVL_PERSIST.stPartsInspection.nHeightDistancePartsGood[3] +1;
GVL_PERSIST.stPartsInspection.nHeightDistanceTotalPartsGood[3] := GVL_PERSIST.stPartsInspection.nHeightDistanceTotalPartsGood[3]+1;
ELSIF GVL_HMI_GLOBAL.aResetHeightSensorGoodParts[3] THEN
GVL_PERSIST.stPartsInspection.nHeightDistancePartsGood[3]:=0;	
END_IF


IF rtrigCaseTriger[11].Q THEN
	GVL_PERSIST.stPartsInspection.nHeightDistancePartsFailed[3]:=GVL_PERSIST.stPartsInspection.nHeightDistancePartsFailed[3] + 1;
	GVL_PERSIST.stPartsInspection.nHeightDistanceTotalPartsFailed[3]:= GVL_PERSIST.stPartsInspection.nHeightDistanceTotalPartsFailed[3] + 1;
ELSIF GVL_HMI_GLOBAL.aResetHeightSensorBadParts[3] THEN
	GVL_PERSIST.stPartsInspection.nHeightDistancePartsFailed[3]:=0;
END_IF
END_ACTION

ACTION ACT_TimTrig:
tonCaseDelay[1](IN:= (stStationStruct.nState=300),PT:=T#50MS);
tonCaseDelay[2](IN:= (stStationStruct.nState=1010),PT:=T#100MS);
tonCaseDelay[3](IN:= (stStationStruct.nState=1240),PT:=T#100MS);
tonCaseDelay[4](IN:= ,PT:=T#1S);
tonCaseDelay[5](IN:=stStationStruct.nState=1220 ,PT:=T#2S);
tonCaseDelay[6](IN:= ,PT:=T#250MS);
tonCaseDelay[7](IN:= ,PT:=T#50MS);
tonCaseDelay[8](IN:= ,PT:=T#250MS);
tonCaseDelay[9](IN:= ,PT:=T#250MS);
tonCaseDelay[10](IN:= ,PT:=T#250MS);

rtrigCaseTriger[1](clk:= );
rtrigCaseTriger[2](clk:= );
rtrigCaseTriger[3](clk:= (stStationStruct.nState=1240) AND GVL_MASTER.stNest.bHeightPass );//
rtrigCaseTriger[4](clk:= (stStationStruct.nState=1240) AND NOT GVL_MASTER.stNest.bHeightPass );//
rtrigCaseTriger[5](clk:= stStationStruct.bStationAbort);
rtrigCaseTriger[6](clk:= (stStationStruct.nState=1240) AND GVL_HMI_GLOBAL.aGeneralPassHeightTest[1]);
rtrigCaseTriger[7](clk:= (stStationStruct.nState=1240) AND GVL_HMI_GLOBAL.aGeneralFailHeightTest[1]);
rtrigCaseTriger[8](clk:= (stStationStruct.nState=1240) AND GVL_HMI_GLOBAL.aGeneralPassHeightTest[2]);
rtrigCaseTriger[9](clk:= (stStationStruct.nState=1240) AND GVL_HMI_GLOBAL.aGeneralFailHeightTest[2]);
rtrigCaseTriger[10](clk:= (stStationStruct.nState=1240) AND GVL_HMI_GLOBAL.aGeneralPassHeightTest[3]);
rtrigCaseTriger[11](clk:= (stStationStruct.nState=1240) AND GVL_HMI_GLOBAL.aGeneralFailHeightTest[3]);
END_ACTION

END_PROGRAM
